QRS_NEXT_CUT()
PTP {E1 29336.909,E2 29336.909}
PTP {X 0,Y 607.909,A -85,B 0,C 180,E1 29336.909,E2 29336.909,E3 0,E4 0,E5 0,E6 0}
QRS_SPEED_INIT()
LIN {X 0,Y 607.909,Z 550,A -85,B 0,C 180,E1 29336.909,E2 29336.909,E3 0,E4 0,E5 0,E6 0} C_VEL
LIN {X 0,Y 607.909,Z 56.154,A -85,B 0,C 180,E1 29336.909,E2 29336.909} C_VEL
LIN {X 0,Y 607.909,Z 48.076,A -85,B 0,C 180,E1 29336.909,E2 29336.909} C_VEL
LIN {X 0,Y 607.891,Z 46.076,A -85,B 0,C 180,E1 29336.721,E2 29336.721} C_VEL
LIN {X 0,Y 607.912,Z 46.07,A -85,B 0,C 180,E1 29333.578,E2 29333.578} C_VEL
LIN {X 0,Y 607.871,Z 46.073,A -85,B 0,C 180,E1 29330.437,E2 29330.437} C_VEL
LIN {X 0,Y 607.918,Z 46.076,A -85,B 0,C 180,E1 29327.268,E2 29327.268} C_VEL
LIN {X 0,Y 607.88,Z 46.071,A -85,B 0,C 180,E1 29324.154,E2 29324.154} C_VEL
LIN {X 0,Y 607.875,Z 46.075,A -85,B 0,C 180,E1 29320.893,E2 29320.893} C_VEL
LIN {X 0,Y 607.917,Z 46.071,A -85,B 0,C 180,E1 29317.772,E2 29317.772} C_VEL
LIN {X 0,Y 607.864,Z 46.073,A -85,B 0,C 180,E1 29314.68,E2 29314.68} C_VEL
LIN {X 0,Y 607.915,Z 46.077,A -85,B 0,C 180,E1 29311.619,E2 29311.619} C_VEL
LIN {X 0,Y 607.867,Z 46.073,A -85,B 0,C 180,E1 29308.572,E2 29308.572} C_VEL
LIN {X 0,Y 607.874,Z 46.076,A -85,B 0,C 180,E1 29305.311,E2 29305.311} C_VEL
LIN {X 0,Y 607.9,Z 46.072,A -85,B 0,C 180,E1 29302.276,E2 29302.276} C_VEL
LIN {X 0,Y 607.858,Z 46.075,A -85,B 0,C 180,E1 29299.167,E2 29299.167} C_VEL
LIN {X 0,Y 607.917,Z 46.075,A -85,B 0,C 180,E1 29296.046,E2 29296.046} C_VEL
LIN {X 0,Y 607.854,Z 46.074,A -85,B 0,C 180,E1 29293.048,E2 29293.048} C_VEL
LIN {X 0,Y 607.895,Z 46.077,A -85,B 0,C 180,E1 29289.9,E2 29289.9} C_VEL
LIN {X 0,Y 607.862,Z 46.075,A -85,B 0,C 180,E1 29286.896,E2 29286.896} C_VEL
LIN {X 0,Y 607.859,Z 46.077,A -85,B 0,C 180,E1 29283.662,E2 29283.662} C_VEL
LIN {X 0,Y 607.917,Z 46.319,A -85,B 0,C 180,E1 29282.298,E2 29282.298} C_VEL
LIN {X 0,Y 607.876,Z 75.31,A -85,B 0,C 180,E1 29279.242,E2 29279.242} C_VEL
LIN {X 0,Y 607.896,Z 105.548,A -85,B 0,C 180,E1 29276.096,E2 29276.096} C_VEL
LIN {X 0,Y 607.888,Z 135.983,A -85,B 0,C 180,E1 29272.993,E2 29272.993} C_VEL
LIN {X 0,Y 607.857,Z 167.849,A -85,B 0,C 180,E1 29269.799,E2 29269.799} C_VEL
LIN {X 0,Y 607.909,Z 175.996,A -85,B 0,C 180,E1 29269.017,E2 29269.017} C_VEL
LIN {X 0,Y 607.889,Z 287.389,A -85,B 0,C 180,E1 29267.665,E2 29267.665} C_VEL
LIN {X 0,Y 607.914,Z 301.952,A -85,B 0,C 180,E1 29267.318,E2 29267.318} C_VEL
LIN {X 0,Y 607.92,Z 316.749,A -85,B 0,C 180,E1 29266.772,E2 29266.772} C_VEL
LIN {X 0,Y 607.887,Z 330.107,A -85,B 0,C 180,E1 29266.089,E2 29266.089} C_VEL
LIN {X 0,Y 607.919,Z 342.573,A -85,B 0,C 180,E1 29265.256,E2 29265.256} C_VEL
LIN {X 0,Y 607.918,Z 354.434,A -85,B 0,C 180,E1 29264.233,E2 29264.233} C_VEL
LIN {X 0,Y 607.918,Z 364.498,A -85,B 0,C 180,E1 29263.118,E2 29263.118} C_VEL
LIN {X 0,Y 607.918,Z 372.672,A -85,B 0,C 180,E1 29261.959,E2 29261.959} C_VEL
LIN {X 0,Y 607.916,Z 379.43,A -85,B 0,C 180,E1 29260.71,E2 29260.71} C_VEL
LIN {X 0,Y 607.917,Z 384.633,A -85,B 0,C 180,E1 29259.37,E2 29259.37} C_VEL
LIN {X 0,Y 607.917,Z 388.043,A -85,B 0,C 180,E1 29258.036,E2 29258.036} C_VEL
LIN {X 0,Y 607.916,Z 389.855,A -85,B 0,C 180,E1 29256.516,E2 29256.516} C_VEL
LIN {X 0,Y 607.916,Z 389.644,A -85,B 0,C 180,E1 29255.095,E2 29255.095} C_VEL
LIN {X 0,Y 607.917,Z 387.832,A -85,B 0,C 180,E1 29253.771,E2 29253.771} C_VEL
LIN {X 0,Y 607.915,Z 384.046,A -85,B 0,C 180,E1 29252.356,E2 29252.356} C_VEL
LIN {X 0,Y 607.916,Z 378.633,A -85,B 0,C 180,E1 29251.036,E2 29251.036} C_VEL
LIN {X 0,Y 607.918,Z 371.814,A -85,B 0,C 180,E1 29249.811,E2 29249.811} C_VEL
LIN {X 0,Y 607.917,Z 362.817,A -85,B 0,C 180,E1 29248.586,E2 29248.586} C_VEL
LIN {X 0,Y 607.919,Z 352.577,A -85,B 0,C 180,E1 29247.501,E2 29247.501} C_VEL
LIN {X 0,Y 607.916,Z 341.267,A -85,B 0,C 180,E1 29246.558,E2 29246.558} C_VEL
LIN {X 0,Y 607.886,Z 328.997,A -85,B 0,C 180,E1 29245.755,E2 29245.755} C_VEL
LIN {X 0,Y 607.919,Z 315.694,A -85,B 0,C 180,E1 29245.093,E2 29245.093} C_VEL
LIN {X 0,Y 607.871,Z 301.315,A -85,B 0,C 180,E1 29244.572,E2 29244.572} C_VEL
LIN {X 0,Y 607.846,Z 285.893,A -85,B 0,C 180,E1 29244.217,E2 29244.217} C_VEL
LIN {X 0,Y 607.887,Z 172.229,A -85,B 0,C 180,E1 29242.842,E2 29242.842} C_VEL
LIN {X 0,Y 607.851,Z 122.898,A -85,B 0,C 180,E1 29239.91,E2 29239.91} C_VEL
LIN {X 0,Y 607.917,Z 72.713,A -85,B 0,C 180,E1 29236.881,E2 29236.881} C_VEL
LIN {X 0,Y 607.911,Z 46.445,A -85,B 0,C 180,E1 29235.248,E2 29235.248} C_VEL
LIN {X 0,Y 607.873,Z 46.078,A -85,B 0,C 180,E1 29234.741,E2 29234.741} C_VEL
LIN {X 0,Y 607.903,Z 46.075,A -85,B 0,C 180,E1 29231.69,E2 29231.69} C_VEL
LIN {X 0,Y 607.917,Z 46.394,A -85,B 0,C 180,E1 29230.67,E2 29230.67} C_VEL
LIN {X 0,Y 607.919,Z 77.534,A -85,B 0,C 180,E1 29228.736,E2 29228.736} C_VEL
LIN {X 0,Y 607.908,Z 131.003,A -85,B 0,C 180,E1 29225.513,E2 29225.513} C_VEL
LIN {X 0,Y 607.913,Z 172.508,A -85,B 0,C 180,E1 29223.057,E2 29223.057} C_VEL
LIN {X 0,Y 607.898,Z 286.479,A -85,B 0,C 180,E1 29221.681,E2 29221.681} C_VEL
LIN {X 0,Y 607.915,Z 301.764,A -85,B 0,C 180,E1 29221.324,E2 29221.324} C_VEL
LIN {X 0,Y 607.919,Z 315.969,A -85,B 0,C 180,E1 29220.805,E2 29220.805} C_VEL
LIN {X 0,Y 607.892,Z 328.884,A -85,B 0,C 180,E1 29220.162,E2 29220.162} C_VEL
LIN {X 0,Y 607.92,Z 342.165,A -85,B 0,C 180,E1 29219.287,E2 29219.287} C_VEL
LIN {X 0,Y 607.918,Z 353.72,A -85,B 0,C 180,E1 29218.301,E2 29218.301} C_VEL
LIN {X 0,Y 607.918,Z 363.5,A -85,B 0,C 180,E1 29217.24,E2 29217.24} C_VEL
LIN {X 0,Y 607.918,Z 371.729,A -85,B 0,C 180,E1 29216.112,E2 29216.112} C_VEL
LIN {X 0,Y 607.918,Z 378.852,A -85,B 0,C 180,E1 29214.829,E2 29214.829} C_VEL
LIN {X 0,Y 607.918,Z 384.09,A -85,B 0,C 180,E1 29213.541,E2 29213.541} C_VEL
LIN {X 0,Y 607.917,Z 387.837,A -85,B 0,C 180,E1 29212.137,E2 29212.137} C_VEL
LIN {X 0,Y 607.919,Z 389.717,A -85,B 0,C 180,E1 29210.712,E2 29210.712} C_VEL
LIN {X 0,Y 607.916,Z 389.794,A -85,B 0,C 180,E1 29209.308,E2 29209.308} C_VEL
LIN {X 0,Y 607.915,Z 388.001,A -85,B 0,C 180,E1 29207.852,E2 29207.852} C_VEL
LIN {X 0,Y 607.915,Z 384.307,A -85,B 0,C 180,E1 29206.438,E2 29206.438} C_VEL
LIN {X 0,Y 607.918,Z 379.055,A -85,B 0,C 180,E1 29205.123,E2 29205.123} C_VEL
LIN {X 0,Y 607.917,Z 371.895,A -85,B 0,C 180,E1 29203.823,E2 29203.823} C_VEL
LIN {X 0,Y 607.918,Z 362.918,A -85,B 0,C 180,E1 29202.598,E2 29202.598} C_VEL
LIN {X 0,Y 607.918,Z 352.733,A -85,B 0,C 180,E1 29201.516,E2 29201.516} C_VEL
LIN {X 0,Y 607.92,Z 341.77,A -85,B 0,C 180,E1 29200.594,E2 29200.594} C_VEL
LIN {X 0,Y 607.916,Z 328.454,A -85,B 0,C 180,E1 29199.724,E2 29199.724} C_VEL
LIN {X 0,Y 607.919,Z 314.572,A -85,B 0,C 180,E1 29199.045,E2 29199.045} C_VEL
LIN {X 0,Y 607.914,Z 300.906,A -85,B 0,C 180,E1 29198.562,E2 29198.562} C_VEL
LIN {X 0,Y 607.908,Z 285.815,A -85,B 0,C 180,E1 29198.217,E2 29198.217} C_VEL
LIN {X 0,Y 607.916,Z 175.701,A -85,B 0,C 180,E1 29196.879,E2 29196.879} C_VEL
LIN {X 0,Y 607.918,Z 143.97,A -85,B 0,C 180,E1 29193.723,E2 29193.723} C_VEL
LIN {X 0,Y 607.892,Z 112.689,A -85,B 0,C 180,E1 29190.547,E2 29190.547} C_VEL
LIN {X 0,Y 607.897,Z 82.49,A -85,B 0,C 180,E1 29187.422,E2 29187.422} C_VEL
LIN {X 0,Y 607.918,Z 53.339,A -85,B 0,C 180,E1 29184.332,E2 29184.332} C_VEL
LIN {X 0,Y 607.901,Z 46.197,A -85,B 0,C 180,E1 29183.507,E2 29183.507} C_VEL
LIN {X 0,Y 607.882,Z 46.072,A -85,B 0,C 180,E1 29180.509,E2 29180.509} C_VEL
LIN {X 0,Y 607.872,Z 46.075,A -85,B 0,C 180,E1 29177.321,E2 29177.321} C_VEL
LIN {X 0,Y 607.918,Z 46.072,A -85,B 0,C 180,E1 29174.186,E2 29174.186} C_VEL
LIN {X 0,Y 607.861,Z 46.074,A -85,B 0,C 180,E1 29171.096,E2 29171.096} C_VEL
LIN {X 0,Y 607.908,Z 46.077,A -85,B 0,C 180,E1 29167.942,E2 29167.942} C_VEL
LIN {X 0,Y 607.867,Z 46.074,A -85,B 0,C 180,E1 29164.907,E2 29164.907} C_VEL
LIN {X 0,Y 607.862,Z 46.076,A -85,B 0,C 180,E1 29161.603,E2 29161.603} C_VEL
LIN {X 0,Y 607.906,Z 46.073,A -85,B 0,C 180,E1 29158.586,E2 29158.586} C_VEL
LIN {X 0,Y 607.852,Z 46.075,A -85,B 0,C 180,E1 29155.472,E2 29155.472} C_VEL
LIN {X 0,Y 607.919,Z 46.077,A -85,B 0,C 180,E1 29152.439,E2 29152.439} C_VEL
LIN {X 0,Y 607.852,Z 46.075,A -85,B 0,C 180,E1 29149.384,E2 29149.384} C_VEL
LIN {X 0,Y 607.876,Z 46.077,A -85,B 0,C 180,E1 29146.202,E2 29146.202} C_VEL
LIN {X 0,Y 607.861,Z 46.075,A -85,B 0,C 180,E1 29143.271,E2 29143.271} C_VEL
LIN {X 0,Y 607.854,Z 46.076,A -85,B 0,C 180,E1 29140.093,E2 29140.093} C_VEL
LIN {X 0,Y 607.88,Z 46.075,A -85,B 0,C 180,E1 29137.159,E2 29137.159} C_VEL
LIN {X 0,Y 607.843,Z 46.077,A -85,B 0,C 180,E1 29134.052,E2 29134.052} C_VEL
LIN {X 0,Y 607.904,Z 46.076,A -85,B 0,C 180,E1 29131.046,E2 29131.046} C_VEL
LIN {X 0,Y 607.837,Z 46.077,A -85,B 0,C 180,E1 29128.017,E2 29128.017} C_VEL
LIN {X 0,Y 607.908,Z 46.077,A -85,B 0,C 180,E1 29124.969,E2 29124.969} C_VEL
LIN {X 0,Y 607.834,Z 46.077,A -85,B 0,C 180,E1 29121.993,E2 29121.993} C_VEL
LIN {X 0,Y 607.871,Z 46.078,A -85,B 0,C 180,E1 29118.857,E2 29118.857} C_VEL
LIN {X 0,Y 607.836,Z 46.077,A -85,B 0,C 180,E1 29116.039,E2 29116.039} C_VEL
LIN {X 0,Y 607.868,Z 46.077,A -85,B 0,C 180,E1 29112.92,E2 29112.92} C_VEL
LIN {X 0,Y 607.842,Z 46.077,A -85,B 0,C 180,E1 29110.103,E2 29110.103} C_VEL
LIN {X 0,Y 607.858,Z 46.076,A -85,B 0,C 180,E1 29106.898,E2 29106.898} C_VEL
LIN {X 0,Y 607.86,Z 46.077,A -85,B 0,C 180,E1 29104.002,E2 29104.002} C_VEL
LIN {X 0,Y 607.849,Z 46.079,A -85,B 0,C 180,E1 29100.835,E2 29100.835} C_VEL
LIN {X 0,Y 607.894,Z 46.318,A -85,B 0,C 180,E1 29099.784,E2 29099.784} C_VEL
LIN {X 0,Y 607.919,Z 52.934,A -85,B 0,C 180,E1 29099.292,E2 29099.292} C_VEL
LIN {X 0,Y 607.902,Z 98.568,A -85,B 0,C 180,E1 29096.208,E2 29096.208} C_VEL
LIN {X 0,Y 607.909,Z 145.038,A -85,B 0,C 180,E1 29093.148,E2 29093.148} C_VEL
LIN {X 0,Y 607.901,Z 157.996,A -85,B 0,C 180,E1 29092.33,E2 29092.33} C_VEL
LIN {X 0,Y 607.917,Z 367.301,A -85,B 0,C 180,E1 29089.705,E2 29089.705} C_VEL
LIN {X 0,Y 607.914,Z 385.58,A -85,B 0,C 180,E1 29089.305,E2 29089.305} C_VEL
LIN {X 0,Y 607.912,Z 404.399,A -85,B 0,C 180,E1 29088.707,E2 29088.707} C_VEL
LIN {X 0,Y 607.915,Z 422.05,A -85,B 0,C 180,E1 29087.963,E2 29087.963} C_VEL
LIN {X 0,Y 607.919,Z 438.783,A -85,B 0,C 180,E1 29087.073,E2 29087.073} C_VEL
LIN {X 0,Y 607.916,Z 454.637,A -85,B 0,C 180,E1 29086.041,E2 29086.041} C_VEL
LIN {X 0,Y 607.917,Z 469.558,A -85,B 0,C 180,E1 29084.868,E2 29084.868} C_VEL
LIN {X 0,Y 607.918,Z 483.217,A -85,B 0,C 180,E1 29083.583,E2 29083.583} C_VEL
LIN {X 0,Y 607.916,Z 495.903,A -85,B 0,C 180,E1 29082.154,E2 29082.154} C_VEL
LIN {X 0,Y 607.912,Z 507.221,A -85,B 0,C 180,E1 29080.616,E2 29080.616} C_VEL
LIN {X 0,Y 607.918,Z 516.986,A -85,B 0,C 180,E1 29078.99,E2 29078.99} C_VEL
LIN {X 0,Y 607.91,Z 524.861,A -85,B 0,C 180,E1 29077.35,E2 29077.35} C_VEL
LIN {X 0,Y 607.907,Z 531.106,A -85,B 0,C 180,E1 29075.664,E2 29075.664} C_VEL
LIN {X 0,Y 607.916,Z 535.871,A -85,B 0,C 180,E1 29073.867,E2 29073.867} C_VEL
LIN {X 0,Y 607.914,Z 538.786,A -85,B 0,C 180,E1 29072.074,E2 29072.074} C_VEL
LIN {X 0,Y 607.907,Z 539.939,A -85,B 0,C 180,E1 29070.283,E2 29070.283} C_VEL
LIN {X 0,Y 607.916,Z 539.348,A -85,B 0,C 180,E1 29068.493,E2 29068.493} C_VEL
LIN {X 0,Y 607.908,Z 537.006,A -85,B 0,C 180,E1 29066.701,E2 29066.701} C_VEL
LIN {X 0,Y 607.916,Z 533.098,A -85,B 0,C 180,E1 29065,E2 29065} C_VEL
LIN {X 0,Y 607.91,Z 527.47,A -85,B 0,C 180,E1 29063.295,E2 29063.295} C_VEL
LIN {X 0,Y 607.915,Z 520.426,A -85,B 0,C 180,E1 29061.679,E2 29061.679} C_VEL
LIN {X 0,Y 607.912,Z 511.514,A -85,B 0,C 180,E1 29060.056,E2 29060.056} C_VEL
LIN {X 0,Y 607.919,Z 501.151,A -85,B 0,C 180,E1 29058.522,E2 29058.522} C_VEL
LIN {X 0,Y 607.917,Z 489.353,A -85,B 0,C 180,E1 29057.076,E2 29057.076} C_VEL
LIN {X 0,Y 607.915,Z 476.098,A -85,B 0,C 180,E1 29055.718,E2 29055.718} C_VEL
LIN {X 0,Y 607.917,Z 461.246,A -85,B 0,C 180,E1 29054.45,E2 29054.45} C_VEL
LIN {X 0,Y 607.918,Z 445.235,A -85,B 0,C 180,E1 29053.322,E2 29053.322} C_VEL
LIN {X 0,Y 607.913,Z 429.047,A -85,B 0,C 180,E1 29052.385,E2 29052.385} C_VEL
LIN {X 0,Y 607.914,Z 412.089,A -85,B 0,C 180,E1 29051.593,E2 29051.593} C_VEL
LIN {X 0,Y 607.914,Z 394.258,A -85,B 0,C 180,E1 29050.946,E2 29050.946} C_VEL
LIN {X 0,Y 607.916,Z 375.204,A -85,B 0,C 180,E1 29050.447,E2 29050.447} C_VEL
LIN {X 0,Y 607.916,Z 355.852,A -85,B 0,C 180,E1 29050.129,E2 29050.129} C_VEL
LIN {X 0,Y 607.897,Z 154.774,A -85,B 0,C 180,E1 29047.622,E2 29047.622} C_VEL
LIN {X 0,Y 607.918,Z 76.627,A -85,B 0,C 180,E1 29044.58,E2 29044.58} C_VEL
LIN {X 0,Y 607.913,Z 46.741,A -85,B 0,C 180,E1 29043.374,E2 29043.374} C_VEL
LIN {X 0,Y 607.903,Z 46.125,A -85,B 0,C 180,E1 29043.215,E2 29043.215} C_VEL
LIN {X 0,Y 607.899,Z 46.073,A -85,B 0,C 180,E1 29040.001,E2 29040.001} C_VEL
LIN {X 0,Y 607.9,Z 46.069,A -85,B 0,C 180,E1 29036.845,E2 29036.845} C_VEL
LIN {X 0,Y 607.911,Z 46.076,A -85,B 0,C 180,E1 29033.578,E2 29033.578} C_VEL
LIN {X 0,Y 607.903,Z 46.071,A -85,B 0,C 180,E1 29030.331,E2 29030.331} C_VEL
LIN {X 0,Y 607.893,Z 46.071,A -85,B 0,C 180,E1 29027.187,E2 29027.187} C_VEL
LIN {X 0,Y 607.916,Z 46.077,A -85,B 0,C 180,E1 29023.954,E2 29023.954} C_VEL
LIN {X 0,Y 607.912,Z 46.068,A -85,B 0,C 180,E1 29020.694,E2 29020.694} C_VEL
LIN {X 0,Y 607.889,Z 46.072,A -85,B 0,C 180,E1 29017.487,E2 29017.487} C_VEL
LIN {X 0,Y 607.908,Z 46.074,A -85,B 0,C 180,E1 29014.343,E2 29014.343} C_VEL
LIN {X 0,Y 607.898,Z 46.069,A -85,B 0,C 180,E1 29011.205,E2 29011.205} C_VEL
LIN {X 0,Y 607.894,Z 46.075,A -85,B 0,C 180,E1 29007.954,E2 29007.954} C_VEL
LIN {X 0,Y 607.908,Z 46.071,A -85,B 0,C 180,E1 29004.787,E2 29004.787} C_VEL
LIN {X 0,Y 607.884,Z 46.072,A -85,B 0,C 180,E1 29001.675,E2 29001.675} C_VEL
LIN {X 0,Y 607.919,Z 46.077,A -85,B 0,C 180,E1 28998.508,E2 28998.508} C_VEL
LIN {X 0,Y 607.916,Z 46.068,A -85,B 0,C 180,E1 28995.257,E2 28995.257} C_VEL
LIN {X 0,Y 607.88,Z 46.073,A -85,B 0,C 180,E1 28992.057,E2 28992.057} C_VEL
LIN {X 0,Y 607.913,Z 46.074,A -85,B 0,C 180,E1 28988.894,E2 28988.894} C_VEL
LIN {X 0,Y 607.887,Z 46.07,A -85,B 0,C 180,E1 28985.758,E2 28985.758} C_VEL
LIN {X 0,Y 607.883,Z 46.075,A -85,B 0,C 180,E1 28982.451,E2 28982.451} C_VEL
LIN {X 0,Y 607.914,Z 46.071,A -85,B 0,C 180,E1 28979.34,E2 28979.34} C_VEL
LIN {X 0,Y 607.891,Z 46.076,A -85,B 0,C 180,E1 28976.721,E2 28976.721} C_VEL
LIN {X 0,Y 606.874,Z 46.2,A -85,B 0,C 180,E1 28975.995,E2 28975.995} C_VEL
LIN {X 0,Y 600.5,Z 46.993,A -85,B 0,C 180,E1 28973.958,E2 28973.958} C_VEL
LIN {X 0,Y 599.976,Z 47.06,A -85,B 0,C 180,E1 28973.428,E2 28973.428} C_VEL
LIN {X 0,Y 599.933,Z 47.061,A -85,B 0,C 180,E1 28970.309,E2 28970.309} C_VEL
LIN {X 0,Y 599.964,Z 47.065,A -85,B 0,C 180,E1 28967.096,E2 28967.096} C_VEL
LIN {X 0,Y 599.96,Z 47.059,A -85,B 0,C 180,E1 28963.94,E2 28963.94} C_VEL
LIN {X 0,Y 599.93,Z 47.063,A -85,B 0,C 180,E1 28960.731,E2 28960.731} C_VEL
LIN {X 0,Y 599.978,Z 47.064,A -85,B 0,C 180,E1 28957.565,E2 28957.565} C_VEL
LIN {X 0,Y 599.933,Z 47.061,A -85,B 0,C 180,E1 28954.427,E2 28954.427} C_VEL
LIN {X 0,Y 599.932,Z 47.063,A -85,B 0,C 180,E1 28951.097,E2 28951.097} C_VEL
LIN {X 0,Y 599.977,Z 47.06,A -85,B 0,C 180,E1 28947.998,E2 28947.998} C_VEL
LIN {X 0,Y 599.921,Z 47.062,A -85,B 0,C 180,E1 28944.9,E2 28944.9} C_VEL
LIN {X 0,Y 599.964,Z 47.066,A -85,B 0,C 180,E1 28941.687,E2 28941.687} C_VEL
LIN {X 0,Y 599.936,Z 47.062,A -85,B 0,C 180,E1 28938.574,E2 28938.574} C_VEL
LIN {X 0,Y 599.922,Z 47.065,A -85,B 0,C 180,E1 28935.368,E2 28935.368} C_VEL
LIN {X 0,Y 599.976,Z 47.062,A -85,B 0,C 180,E1 28932.274,E2 28932.274} C_VEL
LIN {X 0,Y 599.913,Z 47.064,A -85,B 0,C 180,E1 28929.172,E2 28929.172} C_VEL
LIN {X 0,Y 599.961,Z 47.067,A -85,B 0,C 180,E1 28926.034,E2 28926.034} C_VEL
LIN {X 0,Y 599.919,Z 47.067,A -85,B 0,C 180,E1 28923.023,E2 28923.023} C_VEL
LIN {X 0,Y 600.016,Z 47.343,A -85,B 0,C 180,E1 28922.435,E2 28922.435} C_VEL
LIN {X 0,Y 600.181,Z 73.388,A -85,B 0,C 180,E1 28919.764,E2 28919.764} C_VEL
LIN {X 0,Y 600.158,Z 103.091,A -85,B 0,C 180,E1 28916.624,E2 28916.624} C_VEL
LIN {X 0,Y 600.06,Z 133.601,A -85,B 0,C 180,E1 28913.467,E2 28913.467} C_VEL
LIN {X 0,Y 599.995,Z 164.422,A -85,B 0,C 180,E1 28910.331,E2 28910.331} C_VEL
LIN {X 0,Y 600.046,Z 176.097,A -85,B 0,C 180,E1 28909.187,E2 28909.187} C_VEL
LIN {X 0,Y 600.052,Z 287.645,A -85,B 0,C 180,E1 28907.816,E2 28907.816} C_VEL
LIN {X 0,Y 600.057,Z 302.488,A -85,B 0,C 180,E1 28907.452,E2 28907.452} C_VEL
LIN {X 0,Y 600.04,Z 317.043,A -85,B 0,C 180,E1 28906.903,E2 28906.903} C_VEL
LIN {X 0,Y 599.98,Z 330.388,A -85,B 0,C 180,E1 28906.208,E2 28906.208} C_VEL
LIN {X 0,Y 599.984,Z 342.784,A -85,B 0,C 180,E1 28905.364,E2 28905.364} C_VEL
LIN {X 0,Y 599.96,Z 354.596,A -85,B 0,C 180,E1 28904.328,E2 28904.328} C_VEL
LIN {X 0,Y 599.943,Z 364.632,A -85,B 0,C 180,E1 28903.197,E2 28903.197} C_VEL
LIN {X 0,Y 599.929,Z 372.773,A -85,B 0,C 180,E1 28902.023,E2 28902.023} C_VEL
LIN {X 0,Y 599.922,Z 379.505,A -85,B 0,C 180,E1 28900.757,E2 28900.757} C_VEL
LIN {X 0,Y 599.918,Z 384.791,A -85,B 0,C 180,E1 28899.366,E2 28899.366} C_VEL
LIN {X 0,Y 599.917,Z 388.072,A -85,B 0,C 180,E1 28898.047,E2 28898.047} C_VEL
LIN {X 0,Y 599.916,Z 389.865,A -85,B 0,C 180,E1 28896.507,E2 28896.507} C_VEL
LIN {X 0,Y 599.916,Z 389.633,A -85,B 0,C 180,E1 28895.067,E2 28895.067} C_VEL
LIN {X 0,Y 599.916,Z 387.798,A -85,B 0,C 180,E1 28893.726,E2 28893.726} C_VEL
LIN {X 0,Y 599.917,Z 383.997,A -85,B 0,C 180,E1 28892.292,E2 28892.292} C_VEL
LIN {X 0,Y 599.922,Z 378.559,A -85,B 0,C 180,E1 28890.954,E2 28890.954} C_VEL
LIN {X 0,Y 599.932,Z 371.709,A -85,B 0,C 180,E1 28889.713,E2 28889.713} C_VEL
LIN {X 0,Y 599.944,Z 362.694,A -85,B 0,C 180,E1 28888.471,E2 28888.471} C_VEL
LIN {X 0,Y 599.964,Z 352.416,A -85,B 0,C 180,E1 28887.373,E2 28887.373} C_VEL
LIN {X 0,Y 599.981,Z 341.056,A -85,B 0,C 180,E1 28886.416,E2 28886.416} C_VEL
LIN {X 0,Y 599.983,Z 328.728,A -85,B 0,C 180,E1 28885.603,E2 28885.603} C_VEL
LIN {X 0,Y 600.041,Z 315.333,A -85,B 0,C 180,E1 28884.933,E2 28884.933} C_VEL
LIN {X 0,Y 600.017,Z 301.58,A -85,B 0,C 180,E1 28884.429,E2 28884.429} C_VEL
LIN {X 0,Y 600.01,Z 285.975,A -85,B 0,C 180,E1 28884.063,E2 28884.063} C_VEL
LIN {X 0,Y 600.047,Z 172.413,A -85,B 0,C 180,E1 28882.676,E2 28882.676} C_VEL
LIN {X 0,Y 600.081,Z 123.44,A -85,B 0,C 180,E1 28879.73,E2 28879.73} C_VEL
LIN {X 0,Y 600.237,Z 74.053,A -85,B 0,C 180,E1 28876.71,E2 28876.71} C_VEL
LIN {X 0,Y 600.139,Z 48.039,A -85,B 0,C 180,E1 28875.086,E2 28875.086} C_VEL
LIN {X 0,Y 599.953,Z 47.121,A -85,B 0,C 180,E1 28874.93,E2 28874.93} C_VEL
LIN {X 0,Y 599.964,Z 47.065,A -85,B 0,C 180,E1 28871.792,E2 28871.792} C_VEL
LIN {X 0,Y 599.99,Z 47.204,A -85,B 0,C 180,E1 28870.935,E2 28870.935} C_VEL
LIN {X 0,Y 600.288,Z 49.166,A -85,B 0,C 180,E1 28870.743,E2 28870.743} C_VEL
LIN {X 0,Y 600.187,Z 101.17,A -85,B 0,C 180,E1 28867.535,E2 28867.535} C_VEL
LIN {X 0,Y 600.062,Z 154.089,A -85,B 0,C 180,E1 28864.327,E2 28864.327} C_VEL
LIN {X 0,Y 600.108,Z 172.928,A -85,B 0,C 180,E1 28863.222,E2 28863.222} C_VEL
LIN {X 0,Y 600.062,Z 287.429,A -85,B 0,C 180,E1 28861.819,E2 28861.819} C_VEL
LIN {X 0,Y 600.061,Z 301.945,A -85,B 0,C 180,E1 28861.47,E2 28861.47} C_VEL
LIN {X 0,Y 600.039,Z 316.2,A -85,B 0,C 180,E1 28860.939,E2 28860.939} C_VEL
LIN {X 0,Y 599.984,Z 329.601,A -85,B 0,C 180,E1 28860.255,E2 28860.255} C_VEL
LIN {X 0,Y 599.985,Z 342.64,A -85,B 0,C 180,E1 28859.375,E2 28859.375} C_VEL
LIN {X 0,Y 599.96,Z 354.535,A -85,B 0,C 180,E1 28858.334,E2 28858.334} C_VEL
LIN {X 0,Y 599.942,Z 365.113,A -85,B 0,C 180,E1 28857.137,E2 28857.137} C_VEL
LIN {X 0,Y 599.93,Z 373.349,A -85,B 0,C 180,E1 28855.927,E2 28855.927} C_VEL
LIN {X 0,Y 599.923,Z 379.915,A -85,B 0,C 180,E1 28854.667,E2 28854.667} C_VEL
LIN {X 0,Y 599.919,Z 385.157,A -85,B 0,C 180,E1 28853.249,E2 28853.249} C_VEL
LIN {X 0,Y 599.916,Z 388.356,A -85,B 0,C 180,E1 28851.876,E2 28851.876} C_VEL
LIN {X 0,Y 599.916,Z 389.888,A -85,B 0,C 180,E1 28850.456,E2 28850.456} C_VEL
LIN {X 0,Y 599.914,Z 389.554,A -85,B 0,C 180,E1 28848.954,E2 28848.954} C_VEL
LIN {X 0,Y 599.917,Z 387.415,A -85,B 0,C 180,E1 28847.546,E2 28847.546} C_VEL
LIN {X 0,Y 599.919,Z 383.661,A -85,B 0,C 180,E1 28846.192,E2 28846.192} C_VEL
LIN {X 0,Y 599.924,Z 377.654,A -85,B 0,C 180,E1 28844.766,E2 28844.766} C_VEL
LIN {X 0,Y 599.932,Z 370.287,A -85,B 0,C 180,E1 28843.497,E2 28843.497} C_VEL
LIN {X 0,Y 599.947,Z 361.441,A -85,B 0,C 180,E1 28842.323,E2 28842.323} C_VEL
LIN {X 0,Y 599.969,Z 350.727,A -85,B 0,C 180,E1 28841.213,E2 28841.213} C_VEL
LIN {X 0,Y 599.981,Z 338.758,A -85,B 0,C 180,E1 28840.249,E2 28840.249} C_VEL
LIN {X 0,Y 600.014,Z 326.653,A -85,B 0,C 180,E1 28839.488,E2 28839.488} C_VEL
LIN {X 0,Y 600.045,Z 313.017,A -85,B 0,C 180,E1 28838.834,E2 28838.834} C_VEL
LIN {X 0,Y 600.064,Z 297.902,A -85,B 0,C 180,E1 28838.326,E2 28838.326} C_VEL
LIN {X 0,Y 600.076,Z 283.303,A -85,B 0,C 180,E1 28838.024,E2 28838.024} C_VEL
LIN {X 0,Y 600.03,Z 175.769,A -85,B 0,C 180,E1 28836.708,E2 28836.708} C_VEL
LIN {X 0,Y 600.074,Z 144.357,A -85,B 0,C 180,E1 28833.544,E2 28833.544} C_VEL
LIN {X 0,Y 600.127,Z 113.017,A -85,B 0,C 180,E1 28830.32,E2 28830.32} C_VEL
LIN {X 0,Y 600.201,Z 82.376,A -85,B 0,C 180,E1 28827.105,E2 28827.105} C_VEL
LIN {X 0,Y 600.381,Z 53.646,A -85,B 0,C 180,E1 28823.976,E2 28823.976} C_VEL
LIN {X 0,Y 600.154,Z 48.131,A -85,B 0,C 180,E1 28823.36,E2 28823.36} C_VEL
LIN {X 0,Y 599.942,Z 47.125,A -85,B 0,C 180,E1 28823.161,E2 28823.161} C_VEL
LIN {X 0,Y 599.978,Z 47.064,A -85,B 0,C 180,E1 28819.977,E2 28819.977} C_VEL
LIN {X 0,Y 599.927,Z 47.063,A -85,B 0,C 180,E1 28816.858,E2 28816.858} C_VEL
LIN {X 0,Y 599.956,Z 47.066,A -85,B 0,C 180,E1 28813.689,E2 28813.689} C_VEL
LIN {X 0,Y 599.951,Z 47.061,A -85,B 0,C 180,E1 28810.564,E2 28810.564} C_VEL
LIN {X 0,Y 599.922,Z 47.064,A -85,B 0,C 180,E1 28807.373,E2 28807.373} C_VEL
LIN {X 0,Y 599.979,Z 47.063,A -85,B 0,C 180,E1 28804.301,E2 28804.301} C_VEL
LIN {X 0,Y 599.917,Z 47.063,A -85,B 0,C 180,E1 28801.242,E2 28801.242} C_VEL
LIN {X 0,Y 599.957,Z 47.066,A -85,B 0,C 180,E1 28798.09,E2 28798.09} C_VEL
LIN {X 0,Y 599.93,Z 47.063,A -85,B 0,C 180,E1 28795.028,E2 28795.028} C_VEL
LIN {X 0,Y 599.917,Z 47.065,A -85,B 0,C 180,E1 28791.759,E2 28791.759} C_VEL
LIN {X 0,Y 599.978,Z 47.063,A -85,B 0,C 180,E1 28788.659,E2 28788.659} C_VEL
LIN {X 0,Y 599.908,Z 47.064,A -85,B 0,C 180,E1 28785.621,E2 28785.621} C_VEL
LIN {X 0,Y 599.969,Z 47.066,A -85,B 0,C 180,E1 28782.544,E2 28782.544} C_VEL
LIN {X 0,Y 599.911,Z 47.064,A -85,B 0,C 180,E1 28779.5,E2 28779.5} C_VEL
LIN {X 0,Y 599.915,Z 47.066,A -85,B 0,C 180,E1 28776.205,E2 28776.205} C_VEL
LIN {X 0,Y 599.937,Z 47.065,A -85,B 0,C 180,E1 28773.257,E2 28773.257} C_VEL
LIN {X 0,Y 599.901,Z 47.066,A -85,B 0,C 180,E1 28770.11,E2 28770.11} C_VEL
LIN {X 0,Y 599.968,Z 47.066,A -85,B 0,C 180,E1 28767.093,E2 28767.093} C_VEL
LIN {X 0,Y 599.896,Z 47.066,A -85,B 0,C 180,E1 28764.078,E2 28764.078} C_VEL
LIN {X 0,Y 599.963,Z 47.068,A -85,B 0,C 180,E1 28761.076,E2 28761.076} C_VEL
LIN {X 0,Y 599.893,Z 47.067,A -85,B 0,C 180,E1 28758.06,E2 28758.06} C_VEL
LIN {X 0,Y 599.937,Z 47.066,A -85,B 0,C 180,E1 28754.962,E2 28754.962} C_VEL
LIN {X 0,Y 599.902,Z 47.066,A -85,B 0,C 180,E1 28752.068,E2 28752.068} C_VEL
LIN {X 0,Y 599.913,Z 47.066,A -85,B 0,C 180,E1 28748.805,E2 28748.805} C_VEL
LIN {X 0,Y 599.926,Z 47.067,A -85,B 0,C 180,E1 28745.906,E2 28745.906} C_VEL
LIN {X 0,Y 599.909,Z 47.066,A -85,B 0,C 180,E1 28742.798,E2 28742.798} C_VEL
LIN {X 0,Y 599.945,Z 47.264,A -85,B 0,C 180,E1 28740.142,E2 28740.142} C_VEL
LIN {X 0,Y 600.606,Z 50.341,A -85,B 0,C 180,E1 28739.85,E2 28739.85} C_VEL
LIN {X 0,Y 600.513,Z 95.338,A -85,B 0,C 180,E1 28736.774,E2 28736.774} C_VEL
LIN {X 0,Y 600.378,Z 142.596,A -85,B 0,C 180,E1 28733.616,E2 28733.616} C_VEL
LIN {X 0,Y 600.408,Z 158.125,A -85,B 0,C 180,E1 28732.622,E2 28732.622} C_VEL
LIN {X 0,Y 600.377,Z 367.301,A -85,B 0,C 180,E1 28729.963,E2 28729.963} C_VEL
LIN {X 0,Y 600.334,Z 386.274,A -85,B 0,C 180,E1 28729.538,E2 28729.538} C_VEL
LIN {X 0,Y 600.284,Z 404.396,A -85,B 0,C 180,E1 28728.954,E2 28728.954} C_VEL
LIN {X 0,Y 600.23,Z 422.045,A -85,B 0,C 180,E1 28728.201,E2 28728.201} C_VEL
LIN {X 0,Y 600.179,Z 438.697,A -85,B 0,C 180,E1 28727.305,E2 28727.305} C_VEL
LIN {X 0,Y 600.121,Z 454.633,A -85,B 0,C 180,E1 28726.255,E2 28726.255} C_VEL
LIN {X 0,Y 600.069,Z 469.558,A -85,B 0,C 180,E1 28725.067,E2 28725.067} C_VEL
LIN {X 0,Y 600.022,Z 483.015,A -85,B 0,C 180,E1 28723.786,E2 28723.786} C_VEL
LIN {X 0,Y 599.982,Z 495.905,A -85,B 0,C 180,E1 28722.317,E2 28722.317} C_VEL
LIN {X 0,Y 599.954,Z 507.223,A -85,B 0,C 180,E1 28720.758,E2 28720.758} C_VEL
LIN {X 0,Y 599.935,Z 516.988,A -85,B 0,C 180,E1 28719.11,E2 28719.11} C_VEL
LIN {X 0,Y 599.921,Z 525.04,A -85,B 0,C 180,E1 28717.406,E2 28717.406} C_VEL
LIN {X 0,Y 599.911,Z 531.409,A -85,B 0,C 180,E1 28715.644,E2 28715.644} C_VEL
LIN {X 0,Y 599.915,Z 535.872,A -85,B 0,C 180,E1 28713.919,E2 28713.919} C_VEL
LIN {X 0,Y 599.914,Z 538.787,A -85,B 0,C 180,E1 28712.102,E2 28712.102} C_VEL
LIN {X 0,Y 599.907,Z 539.939,A -85,B 0,C 180,E1 28710.287,E2 28710.287} C_VEL
LIN {X 0,Y 599.915,Z 539.349,A -85,B 0,C 180,E1 28708.473,E2 28708.473} C_VEL
LIN {X 0,Y 599.907,Z 537.007,A -85,B 0,C 180,E1 28706.657,E2 28706.657} C_VEL
LIN {X 0,Y 599.917,Z 533.099,A -85,B 0,C 180,E1 28704.933,E2 28704.933} C_VEL
LIN {X 0,Y 599.919,Z 527.47,A -85,B 0,C 180,E1 28703.205,E2 28703.205} C_VEL
LIN {X 0,Y 599.929,Z 520.427,A -85,B 0,C 180,E1 28701.567,E2 28701.567} C_VEL
LIN {X 0,Y 599.942,Z 511.515,A -85,B 0,C 180,E1 28699.923,E2 28699.923} C_VEL
LIN {X 0,Y 599.969,Z 501.152,A -85,B 0,C 180,E1 28698.368,E2 28698.368} C_VEL
LIN {X 0,Y 600.002,Z 489.355,A -85,B 0,C 180,E1 28696.902,E2 28696.902} C_VEL
LIN {X 0,Y 600.046,Z 475.762,A -85,B 0,C 180,E1 28695.494,E2 28695.494} C_VEL
LIN {X 0,Y 600.103,Z 461.244,A -85,B 0,C 180,E1 28694.243,E2 28694.243} C_VEL
LIN {X 0,Y 600.165,Z 445.239,A -85,B 0,C 180,E1 28693.1,E2 28693.1} C_VEL
LIN {X 0,Y 600.219,Z 428.058,A -85,B 0,C 180,E1 28692.102,E2 28692.102} C_VEL
LIN {X 0,Y 600.278,Z 410.698,A -85,B 0,C 180,E1 28691.295,E2 28691.295} C_VEL
LIN {X 0,Y 600.329,Z 392.689,A -85,B 0,C 180,E1 28690.649,E2 28690.649} C_VEL
LIN {X 0,Y 600.368,Z 374.196,A -85,B 0,C 180,E1 28690.172,E2 28690.172} C_VEL
LIN {X 0,Y 600.391,Z 354.456,A -85,B 0,C 180,E1 28689.852,E2 28689.852} C_VEL
LIN {X 0,Y 600.442,Z 154.702,A -85,B 0,C 180,E1 28687.327,E2 28687.327} C_VEL
LIN {X 0,Y 600.604,Z 75.307,A -85,B 0,C 180,E1 28684.195,E2 28684.195} C_VEL
LIN {X 0,Y 600.647,Z 49.473,A -85,B 0,C 180,E1 28683.157,E2 28683.157} C_VEL
LIN {X 0,Y 600.013,Z 47.428,A -85,B 0,C 180,E1 28683,E2 28683} C_VEL
LIN {X 0,Y 599.973,Z 47.062,A -85,B 0,C 180,E1 28682.402,E2 28682.402} C_VEL
LIN {X 0,Y 599.958,Z 47.062,A -85,B 0,C 180,E1 28679.123,E2 28679.123} C_VEL
LIN {X 0,Y 599.964,Z 47.063,A -85,B 0,C 180,E1 28675.921,E2 28675.921} C_VEL
LIN {X 0,Y 599.973,Z 47.057,A -85,B 0,C 180,E1 28672.648,E2 28672.648} C_VEL
LIN {X 0,Y 599.959,Z 47.063,A -85,B 0,C 180,E1 28669.459,E2 28669.459} C_VEL
LIN {X 0,Y 599.965,Z 47.062,A -85,B 0,C 180,E1 28666.244,E2 28666.244} C_VEL
LIN {X 0,Y 599.958,Z 47.059,A -85,B 0,C 180,E1 28663.101,E2 28663.101} C_VEL
LIN {X 0,Y 599.963,Z 47.064,A -85,B 0,C 180,E1 28659.788,E2 28659.788} C_VEL
LIN {X 0,Y 599.966,Z 47.06,A -85,B 0,C 180,E1 28656.56,E2 28656.56} C_VEL
LIN {X 0,Y 599.951,Z 47.06,A -85,B 0,C 180,E1 28653.392,E2 28653.392} C_VEL
LIN {X 0,Y 599.97,Z 47.066,A -85,B 0,C 180,E1 28650.129,E2 28650.129} C_VEL
LIN {X 0,Y 599.971,Z 47.058,A -85,B 0,C 180,E1 28646.848,E2 28646.848} C_VEL
LIN {X 0,Y 599.945,Z 47.06,A -85,B 0,C 180,E1 28643.681,E2 28643.681} C_VEL
LIN {X 0,Y 599.978,Z 47.066,A -85,B 0,C 180,E1 28640.485,E2 28640.485} C_VEL
LIN {X 0,Y 599.978,Z 47.057,A -85,B 0,C 180,E1 28637.156,E2 28637.156} C_VEL
LIN {X 0,Y 599.942,Z 47.062,A -85,B 0,C 180,E1 28633.984,E2 28633.984} C_VEL
LIN {X 0,Y 599.975,Z 47.065,A -85,B 0,C 180,E1 28630.757,E2 28630.757} C_VEL
LIN {X 0,Y 599.968,Z 47.058,A -85,B 0,C 180,E1 28627.469,E2 28627.469} C_VEL
LIN {X 0,Y 599.941,Z 47.062,A -85,B 0,C 180,E1 28624.301,E2 28624.301} C_VEL
LIN {X 0,Y 599.974,Z 47.062,A -85,B 0,C 180,E1 28621.146,E2 28621.146} C_VEL
LIN {X 0,Y 599.941,Z 47.06,A -85,B 0,C 180,E1 28617.994,E2 28617.994} C_VEL
LIN {X 0,Y 599.95,Z 47.064,A -85,B 0,C 180,E1 28614.741,E2 28614.741} C_VEL
LIN {X 0,Y 599.976,Z 47.06,A -85,B 0,C 180,E1 28613.428,E2 28613.428} C_VEL
LIN {X 0,Y 598.978,Z 47.191,A -85,B 0,C 180,E1 28612.693,E2 28612.693} C_VEL
LIN {X 0,Y 592.517,Z 47.988,A -85,B 0,C 180,E1 28610.629,E2 28610.629} C_VEL
LIN {X 0,Y 592.003,Z 48.049,A -85,B 0,C 180,E1 28610.092,E2 28610.092} C_VEL
LIN {X 0,Y 592.003,Z 48.052,A -85,B 0,C 180,E1 28606.82,E2 28606.82} C_VEL
LIN {X 0,Y 592.038,Z 48.05,A -85,B 0,C 180,E1 28603.618,E2 28603.618} C_VEL
LIN {X 0,Y 591.991,Z 48.051,A -85,B 0,C 180,E1 28600.462,E2 28600.462} C_VEL
LIN {X 0,Y 592.017,Z 48.051,A -85,B 0,C 180,E1 28597.237,E2 28597.237} C_VEL
LIN {X 0,Y 592.025,Z 48.048,A -85,B 0,C 180,E1 28594.06,E2 28594.06} C_VEL
LIN {X 0,Y 591.985,Z 48.051,A -85,B 0,C 180,E1 28590.831,E2 28590.831} C_VEL
LIN {X 0,Y 592.036,Z 48.054,A -85,B 0,C 180,E1 28587.745,E2 28587.745} C_VEL
LIN {X 0,Y 591.991,Z 48.05,A -85,B 0,C 180,E1 28584.597,E2 28584.597} C_VEL
LIN {X 0,Y 591.989,Z 48.053,A -85,B 0,C 180,E1 28581.287,E2 28581.287} C_VEL
LIN {X 0,Y 592.035,Z 48.051,A -85,B 0,C 180,E1 28578.138,E2 28578.138} C_VEL
LIN {X 0,Y 591.978,Z 48.053,A -85,B 0,C 180,E1 28575.046,E2 28575.046} C_VEL
LIN {X 0,Y 592.017,Z 48.055,A -85,B 0,C 180,E1 28571.857,E2 28571.857} C_VEL
LIN {X 0,Y 591.99,Z 48.053,A -85,B 0,C 180,E1 28568.799,E2 28568.799} C_VEL
LIN {X 0,Y 591.977,Z 48.055,A -85,B 0,C 180,E1 28565.521,E2 28565.521} C_VEL
LIN {X 0,Y 592.052,Z 48.282,A -85,B 0,C 180,E1 28562.596,E2 28562.596} C_VEL
LIN {X 0,Y 592.318,Z 55.545,A -85,B 0,C 180,E1 28561.843,E2 28561.843} C_VEL
LIN {X 0,Y 592.462,Z 87.287,A -85,B 0,C 180,E1 28558.582,E2 28558.582} C_VEL
LIN {X 0,Y 592.334,Z 117.062,A -85,B 0,C 180,E1 28555.433,E2 28555.433} C_VEL
LIN {X 0,Y 592.188,Z 148.276,A -85,B 0,C 180,E1 28552.185,E2 28552.185} C_VEL
LIN {X 0,Y 592.124,Z 175.848,A -85,B 0,C 180,E1 28549.377,E2 28549.377} C_VEL
LIN {X 0,Y 592.316,Z 202.602,A -85,B 0,C 180,E1 28549.034,E2 28549.034} C_VEL
LIN {X 0,Y 592.22,Z 287.638,A -85,B 0,C 180,E1 28547.975,E2 28547.975} C_VEL
LIN {X 0,Y 592.207,Z 302.133,A -85,B 0,C 180,E1 28547.617,E2 28547.617} C_VEL
LIN {X 0,Y 592.166,Z 316.288,A -85,B 0,C 180,E1 28547.084,E2 28547.084} C_VEL
LIN {X 0,Y 592.079,Z 329.845,A -85,B 0,C 180,E1 28546.38,E2 28546.38} C_VEL
LIN {X 0,Y 592.051,Z 342.344,A -85,B 0,C 180,E1 28545.525,E2 28545.525} C_VEL
LIN {X 0,Y 592.008,Z 353.754,A -85,B 0,C 180,E1 28544.524,E2 28544.524} C_VEL
LIN {X 0,Y 591.971,Z 363.19,A -85,B 0,C 180,E1 28543.478,E2 28543.478} C_VEL
LIN {X 0,Y 591.944,Z 371.672,A -85,B 0,C 180,E1 28542.287,E2 28542.287} C_VEL
LIN {X 0,Y 591.927,Z 378.659,A -85,B 0,C 180,E1 28541.003,E2 28541.003} C_VEL
LIN {X 0,Y 591.92,Z 384.129,A -85,B 0,C 180,E1 28539.626,E2 28539.626} C_VEL
LIN {X 0,Y 591.917,Z 387.916,A -85,B 0,C 180,E1 28538.156,E2 28538.156} C_VEL
LIN {X 0,Y 591.916,Z 389.766,A -85,B 0,C 180,E1 28536.661,E2 28536.661} C_VEL
LIN {X 0,Y 591.916,Z 389.755,A -85,B 0,C 180,E1 28535.233,E2 28535.233} C_VEL
LIN {X 0,Y 591.916,Z 387.965,A -85,B 0,C 180,E1 28533.776,E2 28533.776} C_VEL
LIN {X 0,Y 591.918,Z 384.248,A -85,B 0,C 180,E1 28532.323,E2 28532.323} C_VEL
LIN {X 0,Y 591.927,Z 378.943,A -85,B 0,C 180,E1 28530.967,E2 28530.967} C_VEL
LIN {X 0,Y 591.945,Z 372.211,A -85,B 0,C 180,E1 28529.709,E2 28529.709} C_VEL
LIN {X 0,Y 591.97,Z 363.338,A -85,B 0,C 180,E1 28528.451,E2 28528.451} C_VEL
LIN {X 0,Y 592.008,Z 353.752,A -85,B 0,C 180,E1 28527.386,E2 28527.386} C_VEL
LIN {X 0,Y 592.052,Z 342.125,A -85,B 0,C 180,E1 28526.368,E2 28526.368} C_VEL
LIN {X 0,Y 592.079,Z 329.438,A -85,B 0,C 180,E1 28525.505,E2 28525.505} C_VEL
LIN {X 0,Y 592.166,Z 316.078,A -85,B 0,C 180,E1 28524.817,E2 28524.817} C_VEL
LIN {X 0,Y 592.165,Z 301.823,A -85,B 0,C 180,E1 28524.282,E2 28524.282} C_VEL
LIN {X 0,Y 592.178,Z 286.584,A -85,B 0,C 180,E1 28523.914,E2 28523.914} C_VEL
LIN {X 0,Y 592.196,Z 172.307,A -85,B 0,C 180,E1 28522.493,E2 28522.493} C_VEL
LIN {X 0,Y 592.324,Z 123.182,A -85,B 0,C 180,E1 28519.495,E2 28519.495} C_VEL
LIN {X 0,Y 592.569,Z 73.804,A -85,B 0,C 180,E1 28516.435,E2 28516.435} C_VEL
LIN {X 0,Y 592.502,Z 50.051,A -85,B 0,C 180,E1 28514.937,E2 28514.937} C_VEL
LIN {X 0,Y 592.02,Z 48.234,A -85,B 0,C 180,E1 28514.755,E2 28514.755} C_VEL
LIN {X 0,Y 592.025,Z 48.053,A -85,B 0,C 180,E1 28511.691,E2 28511.691} C_VEL
LIN {X 0,Y 592.08,Z 48.368,A -85,B 0,C 180,E1 28511.131,E2 28511.131} C_VEL
LIN {X 0,Y 592.664,Z 51.639,A -85,B 0,C 180,E1 28510.867,E2 28510.867} C_VEL
LIN {X 0,Y 592.453,Z 103.221,A -85,B 0,C 180,E1 28507.645,E2 28507.645} C_VEL
LIN {X 0,Y 592.24,Z 156.193,A -85,B 0,C 180,E1 28504.393,E2 28504.393} C_VEL
LIN {X 0,Y 592.243,Z 172.5,A -85,B 0,C 180,E1 28503.41,E2 28503.41} C_VEL
LIN {X 0,Y 592.228,Z 287.359,A -85,B 0,C 180,E1 28501.979,E2 28501.979} C_VEL
LIN {X 0,Y 592.213,Z 301.992,A -85,B 0,C 180,E1 28501.623,E2 28501.623} C_VEL
LIN {X 0,Y 592.165,Z 316.211,A -85,B 0,C 180,E1 28501.087,E2 28501.087} C_VEL
LIN {X 0,Y 592.086,Z 329.119,A -85,B 0,C 180,E1 28500.423,E2 28500.423} C_VEL
LIN {X 0,Y 592.059,Z 342.262,A -85,B 0,C 180,E1 28499.532,E2 28499.532} C_VEL
LIN {X 0,Y 592.007,Z 354.099,A -85,B 0,C 180,E1 28498.49,E2 28498.49} C_VEL
LIN {X 0,Y 591.969,Z 363.819,A -85,B 0,C 180,E1 28497.398,E2 28497.398} C_VEL
LIN {X 0,Y 591.942,Z 372.171,A -85,B 0,C 180,E1 28496.207,E2 28496.207} C_VEL
LIN {X 0,Y 591.928,Z 379.47,A -85,B 0,C 180,E1 28494.83,E2 28494.83} C_VEL
LIN {X 0,Y 591.919,Z 384.468,A -85,B 0,C 180,E1 28493.516,E2 28493.516} C_VEL
LIN {X 0,Y 591.918,Z 388.1,A -85,B 0,C 180,E1 28492.058,E2 28492.058} C_VEL
LIN {X 0,Y 591.917,Z 389.856,A -85,B 0,C 180,E1 28490.531,E2 28490.531} C_VEL
LIN {X 0,Y 591.916,Z 389.618,A -85,B 0,C 180,E1 28489.032,E2 28489.032} C_VEL
LIN {X 0,Y 591.917,Z 387.65,A -85,B 0,C 180,E1 28487.624,E2 28487.624} C_VEL
LIN {X 0,Y 591.92,Z 383.729,A -85,B 0,C 180,E1 28486.161,E2 28486.161} C_VEL
LIN {X 0,Y 591.93,Z 378.052,A -85,B 0,C 180,E1 28484.78,E2 28484.78} C_VEL
LIN {X 0,Y 591.946,Z 370.95,A -85,B 0,C 180,E1 28483.511,E2 28483.511} C_VEL
LIN {X 0,Y 591.976,Z 362.018,A -85,B 0,C 180,E1 28482.286,E2 28482.286} C_VEL
LIN {X 0,Y 592.018,Z 351.076,A -85,B 0,C 180,E1 28481.127,E2 28481.127} C_VEL
LIN {X 0,Y 592.058,Z 338.973,A -85,B 0,C 180,E1 28480.133,E2 28480.133} C_VEL
LIN {X 0,Y 592.118,Z 326.554,A -85,B 0,C 180,E1 28479.341,E2 28479.341} C_VEL
LIN {X 0,Y 592.18,Z 312.482,A -85,B 0,C 180,E1 28478.662,E2 28478.662} C_VEL
LIN {X 0,Y 592.223,Z 296.996,A -85,B 0,C 180,E1 28478.144,E2 28478.144} C_VEL
LIN {X 0,Y 592.25,Z 281.762,A -85,B 0,C 180,E1 28477.841,E2 28477.841} C_VEL
LIN {X 0,Y 592.151,Z 176.009,A -85,B 0,C 180,E1 28476.538,E2 28476.538} C_VEL
LIN {X 0,Y 592.232,Z 145.962,A -85,B 0,C 180,E1 28473.487,E2 28473.487} C_VEL
LIN {X 0,Y 592.351,Z 114.424,A -85,B 0,C 180,E1 28470.2,E2 28470.2} C_VEL
LIN {X 0,Y 592.523,Z 85.445,A -85,B 0,C 180,E1 28467.105,E2 28467.105} C_VEL
LIN {X 0,Y 592.837,Z 56.662,A -85,B 0,C 180,E1 28463.92,E2 28463.92} C_VEL
LIN {X 0,Y 592.66,Z 50.727,A -85,B 0,C 180,E1 28463.252,E2 28463.252} C_VEL
LIN {X 0,Y 592.001,Z 48.143,A -85,B 0,C 180,E1 28462.885,E2 28462.885} C_VEL
LIN {X 0,Y 592.035,Z 48.055,A -85,B 0,C 180,E1 28459.741,E2 28459.741} C_VEL
LIN {X 0,Y 592.003,Z 48.051,A -85,B 0,C 180,E1 28456.585,E2 28456.585} C_VEL
LIN {X 0,Y 591.992,Z 48.054,A -85,B 0,C 180,E1 28453.379,E2 28453.379} C_VEL
LIN {X 0,Y 592.039,Z 48.051,A -85,B 0,C 180,E1 28450.214,E2 28450.214} C_VEL
LIN {X 0,Y 591.983,Z 48.052,A -85,B 0,C 180,E1 28447.083,E2 28447.083} C_VEL
LIN {X 0,Y 592.01,Z 48.055,A -85,B 0,C 180,E1 28443.874,E2 28443.874} C_VEL
LIN {X 0,Y 592.006,Z 48.051,A -85,B 0,C 180,E1 28440.774,E2 28440.774} C_VEL
LIN {X 0,Y 591.978,Z 48.054,A -85,B 0,C 180,E1 28437.58,E2 28437.58} C_VEL
LIN {X 0,Y 592.041,Z 48.053,A -85,B 0,C 180,E1 28434.476,E2 28434.476} C_VEL
LIN {X 0,Y 591.975,Z 48.053,A -85,B 0,C 180,E1 28431.355,E2 28431.355} C_VEL
LIN {X 0,Y 591.994,Z 48.055,A -85,B 0,C 180,E1 28428.109,E2 28428.109} C_VEL
LIN {X 0,Y 591.994,Z 48.052,A -85,B 0,C 180,E1 28425.124,E2 28425.124} C_VEL
LIN {X 0,Y 591.97,Z 48.054,A -85,B 0,C 180,E1 28421.894,E2 28421.894} C_VEL
LIN {X 0,Y 592.037,Z 48.054,A -85,B 0,C 180,E1 28418.787,E2 28418.787} C_VEL
LIN {X 0,Y 591.964,Z 48.054,A -85,B 0,C 180,E1 28415.768,E2 28415.768} C_VEL
LIN {X 0,Y 592.011,Z 48.055,A -85,B 0,C 180,E1 28412.653,E2 28412.653} C_VEL
LIN {X 0,Y 591.968,Z 48.055,A -85,B 0,C 180,E1 28409.666,E2 28409.666} C_VEL
LIN {X 0,Y 591.967,Z 48.055,A -85,B 0,C 180,E1 28406.358,E2 28406.358} C_VEL
LIN {X 0,Y 591.998,Z 48.055,A -85,B 0,C 180,E1 28403.402,E2 28403.402} C_VEL
LIN {X 0,Y 591.957,Z 48.056,A -85,B 0,C 180,E1 28400.322,E2 28400.322} C_VEL
LIN {X 0,Y 592.028,Z 48.056,A -85,B 0,C 180,E1 28397.278,E2 28397.278} C_VEL
LIN {X 0,Y 591.957,Z 48.056,A -85,B 0,C 180,E1 28394.234,E2 28394.234} C_VEL
LIN {X 0,Y 592.004,Z 48.055,A -85,B 0,C 180,E1 28391.071,E2 28391.071} C_VEL
LIN {X 0,Y 591.964,Z 48.056,A -85,B 0,C 180,E1 28388.184,E2 28388.184} C_VEL
LIN {X 0,Y 591.981,Z 48.056,A -85,B 0,C 180,E1 28384.93,E2 28384.93} C_VEL
LIN {X 0,Y 591.986,Z 48.056,A -85,B 0,C 180,E1 28382.019,E2 28382.019} C_VEL
LIN {X 0,Y 591.999,Z 48.3,A -85,B 0,C 180,E1 28380.472,E2 28380.472} C_VEL
LIN {X 0,Y 593.247,Z 53,A -85,B 0,C 180,E1 28380.038,E2 28380.038} C_VEL
LIN {X 0,Y 593.12,Z 96.992,A -85,B 0,C 180,E1 28377.021,E2 28377.021} C_VEL
LIN {X 0,Y 592.849,Z 145.038,A -85,B 0,C 180,E1 28373.771,E2 28373.771} C_VEL
LIN {X 0,Y 592.863,Z 158.178,A -85,B 0,C 180,E1 28372.925,E2 28372.925} C_VEL
LIN {X 0,Y 593.101,Z 171.968,A -85,B 0,C 180,E1 28372.735,E2 28372.735} C_VEL
LIN {X 0,Y 592.851,Z 367.301,A -85,B 0,C 180,E1 28370.227,E2 28370.227} C_VEL
LIN {X 0,Y 592.771,Z 386.296,A -85,B 0,C 180,E1 28369.797,E2 28369.797} C_VEL
LIN {X 0,Y 592.675,Z 404.393,A -85,B 0,C 180,E1 28369.207,E2 28369.207} C_VEL
LIN {X 0,Y 592.565,Z 422.04,A -85,B 0,C 180,E1 28368.444,E2 28368.444} C_VEL
LIN {X 0,Y 592.459,Z 438.691,A -85,B 0,C 180,E1 28367.538,E2 28367.538} C_VEL
LIN {X 0,Y 592.341,Z 454.63,A -85,B 0,C 180,E1 28366.474,E2 28366.474} C_VEL
LIN {X 0,Y 592.23,Z 469.556,A -85,B 0,C 180,E1 28365.271,E2 28365.271} C_VEL
LIN {X 0,Y 592.136,Z 483.015,A -85,B 0,C 180,E1 28363.974,E2 28363.974} C_VEL
LIN {X 0,Y 592.056,Z 495.422,A -85,B 0,C 180,E1 28362.546,E2 28362.546} C_VEL
LIN {X 0,Y 592,Z 506.585,A -85,B 0,C 180,E1 28361.003,E2 28361.003} C_VEL
LIN {X 0,Y 591.955,Z 516.472,A -85,B 0,C 180,E1 28359.332,E2 28359.332} C_VEL
LIN {X 0,Y 591.935,Z 524.771,A -85,B 0,C 180,E1 28357.571,E2 28357.571} C_VEL
LIN {X 0,Y 591.918,Z 531.25,A -85,B 0,C 180,E1 28355.772,E2 28355.772} C_VEL
LIN {X 0,Y 591.915,Z 535.873,A -85,B 0,C 180,E1 28353.972,E2 28353.972} C_VEL
LIN {X 0,Y 591.913,Z 538.788,A -85,B 0,C 180,E1 28352.13,E2 28352.13} C_VEL
LIN {X 0,Y 591.907,Z 539.939,A -85,B 0,C 180,E1 28350.291,E2 28350.291} C_VEL
LIN {X 0,Y 591.914,Z 539.35,A -85,B 0,C 180,E1 28348.452,E2 28348.452} C_VEL
LIN {X 0,Y 591.907,Z 537.008,A -85,B 0,C 180,E1 28346.611,E2 28346.611} C_VEL
LIN {X 0,Y 591.919,Z 533.1,A -85,B 0,C 180,E1 28344.864,E2 28344.864} C_VEL
LIN {X 0,Y 591.93,Z 527.47,A -85,B 0,C 180,E1 28343.113,E2 28343.113} C_VEL
LIN {X 0,Y 591.943,Z 520.428,A -85,B 0,C 180,E1 28341.453,E2 28341.453} C_VEL
LIN {X 0,Y 591.977,Z 511.517,A -85,B 0,C 180,E1 28339.786,E2 28339.786} C_VEL
LIN {X 0,Y 592.024,Z 501.154,A -85,B 0,C 180,E1 28338.209,E2 28338.209} C_VEL
LIN {X 0,Y 592.094,Z 489.356,A -85,B 0,C 180,E1 28336.724,E2 28336.724} C_VEL
LIN {X 0,Y 592.192,Z 475.589,A -85,B 0,C 180,E1 28335.28,E2 28335.28} C_VEL
LIN {X 0,Y 592.306,Z 460.611,A -85,B 0,C 180,E1 28333.979,E2 28333.979} C_VEL
LIN {X 0,Y 592.422,Z 444.44,A -85,B 0,C 180,E1 28332.822,E2 28332.822} C_VEL
LIN {X 0,Y 592.535,Z 428.063,A -85,B 0,C 180,E1 28331.862,E2 28331.862} C_VEL
LIN {X 0,Y 592.649,Z 411.154,A -85,B 0,C 180,E1 28331.063,E2 28331.063} C_VEL
LIN {X 0,Y 592.752,Z 392.874,A -85,B 0,C 180,E1 28330.397,E2 28330.397} C_VEL
LIN {X 0,Y 592.831,Z 374.359,A -85,B 0,C 180,E1 28329.912,E2 28329.912} C_VEL
LIN {X 0,Y 592.88,Z 354.558,A -85,B 0,C 180,E1 28329.587,E2 28329.587} C_VEL
LIN {X 0,Y 593,Z 155.102,A -85,B 0,C 180,E1 28327.038,E2 28327.038} C_VEL
LIN {X 0,Y 593.308,Z 75.967,A -85,B 0,C 180,E1 28323.88,E2 28323.88} C_VEL
LIN {X 0,Y 593.183,Z 51.428,A -85,B 0,C 180,E1 28322.872,E2 28322.872} C_VEL
LIN {X 0,Y 592.09,Z 48.462,A -85,B 0,C 180,E1 28322.654,E2 28322.654} C_VEL
LIN {X 0,Y 592.027,Z 48.054,A -85,B 0,C 180,E1 28322.218,E2 28322.218} C_VEL
LIN {X 0,Y 592.019,Z 48.05,A -85,B 0,C 180,E1 28318.996,E2 28318.996} C_VEL
LIN {X 0,Y 592.031,Z 48.053,A -85,B 0,C 180,E1 28315.78,E2 28315.78} C_VEL
LIN {X 0,Y 592.03,Z 48.047,A -85,B 0,C 180,E1 28312.435,E2 28312.435} C_VEL
LIN {X 0,Y 592.017,Z 48.051,A -85,B 0,C 180,E1 28309.316,E2 28309.316} C_VEL
LIN {X 0,Y 592.027,Z 48.052,A -85,B 0,C 180,E1 28306.149,E2 28306.149} C_VEL
LIN {X 0,Y 592.034,Z 48.046,A -85,B 0,C 180,E1 28302.867,E2 28302.867} C_VEL
LIN {X 0,Y 592.017,Z 48.052,A -85,B 0,C 180,E1 28299.636,E2 28299.636} C_VEL
LIN {X 0,Y 592.028,Z 48.05,A -85,B 0,C 180,E1 28296.476,E2 28296.476} C_VEL
LIN {X 0,Y 592.018,Z 48.048,A -85,B 0,C 180,E1 28293.282,E2 28293.282} C_VEL
LIN {X 0,Y 592.02,Z 48.053,A -85,B 0,C 180,E1 28289.96,E2 28289.96} C_VEL
LIN {X 0,Y 592.031,Z 48.048,A -85,B 0,C 180,E1 28286.803,E2 28286.803} C_VEL
LIN {X 0,Y 592.008,Z 48.048,A -85,B 0,C 180,E1 28283.595,E2 28283.595} C_VEL
LIN {X 0,Y 592.032,Z 48.054,A -85,B 0,C 180,E1 28280.359,E2 28280.359} C_VEL
LIN {X 0,Y 592.037,Z 48.047,A -85,B 0,C 180,E1 28277.088,E2 28277.088} C_VEL
LIN {X 0,Y 592.004,Z 48.049,A -85,B 0,C 180,E1 28273.876,E2 28273.876} C_VEL
LIN {X 0,Y 592.032,Z 48.054,A -85,B 0,C 180,E1 28270.608,E2 28270.608} C_VEL
LIN {X 0,Y 592.034,Z 48.047,A -85,B 0,C 180,E1 28267.374,E2 28267.374} C_VEL
LIN {X 0,Y 592,Z 48.05,A -85,B 0,C 180,E1 28264.165,E2 28264.165} C_VEL
LIN {X 0,Y 592.039,Z 48.054,A -85,B 0,C 180,E1 28260.967,E2 28260.967} C_VEL
LIN {X 0,Y 592.025,Z 48.047,A -85,B 0,C 180,E1 28257.677,E2 28257.677} C_VEL
LIN {X 0,Y 591.998,Z 48.052,A -85,B 0,C 180,E1 28254.475,E2 28254.475} C_VEL
LIN {X 0,Y 592.036,Z 48.051,A -85,B 0,C 180,E1 28251.355,E2 28251.355} C_VEL
LIN {X 0,Y 592.003,Z 48.049,A -85,B 0,C 180,E1 28250.092,E2 28250.092} C_VEL
LIN {X 0,Y 591.043,Z 48.176,A -85,B 0,C 180,E1 28249.346,E2 28249.346} C_VEL
LIN {X 0,Y 584.513,Z 48.992,A -85,B 0,C 180,E1 28247.2,E2 28247.2} C_VEL
LIN {X 0,Y 584.058,Z 49.04,A -85,B 0,C 180,E1 28246.709,E2 28246.709} C_VEL
LIN {X 0,Y 584.099,Z 49.041,A -85,B 0,C 180,E1 28243.491,E2 28243.491} C_VEL
LIN {X 0,Y 584.059,Z 49.039,A -85,B 0,C 180,E1 28240.29,E2 28240.29} C_VEL
LIN {X 0,Y 584.055,Z 49.038,A -85,B 0,C 180,E1 28236.919,E2 28236.919} C_VEL
LIN {X 0,Y 584.1,Z 49.039,A -85,B 0,C 180,E1 28233.76,E2 28233.76} C_VEL
LIN {X 0,Y 584.05,Z 49.038,A -85,B 0,C 180,E1 28230.572,E2 28230.572} C_VEL
LIN {X 0,Y 584.058,Z 49.043,A -85,B 0,C 180,E1 28227.25,E2 28227.25} C_VEL
LIN {X 0,Y 584.097,Z 49.038,A -85,B 0,C 180,E1 28224.062,E2 28224.062} C_VEL
LIN {X 0,Y 584.042,Z 49.041,A -85,B 0,C 180,E1 28220.949,E2 28220.949} C_VEL
LIN {X 0,Y 584.079,Z 49.044,A -85,B 0,C 180,E1 28217.719,E2 28217.719} C_VEL
LIN {X 0,Y 584.054,Z 49.041,A -85,B 0,C 180,E1 28214.715,E2 28214.715} C_VEL
LIN {X 0,Y 584.041,Z 49.043,A -85,B 0,C 180,E1 28211.423,E2 28211.423} C_VEL
LIN {X 0,Y 584.097,Z 49.043,A -85,B 0,C 180,E1 28208.29,E2 28208.29} C_VEL
LIN {X 0,Y 584.035,Z 49.044,A -85,B 0,C 180,E1 28205.234,E2 28205.234} C_VEL
LIN {X 0,Y 584.103,Z 49.316,A -85,B 0,C 180,E1 28202.745,E2 28202.745} C_VEL
LIN {X 0,Y 584.509,Z 53.251,A -85,B 0,C 180,E1 28202.324,E2 28202.324} C_VEL
LIN {X 0,Y 584.687,Z 83.63,A -85,B 0,C 180,E1 28199.223,E2 28199.223} C_VEL
LIN {X 0,Y 584.601,Z 112.552,A -85,B 0,C 180,E1 28196.183,E2 28196.183} C_VEL
LIN {X 0,Y 584.408,Z 144.038,A -85,B 0,C 180,E1 28192.852,E2 28192.852} C_VEL
LIN {X 0,Y 584.206,Z 175.491,A -85,B 0,C 180,E1 28189.585,E2 28189.585} C_VEL
LIN {X 0,Y 584.545,Z 180.922,A -85,B 0,C 180,E1 28189.48,E2 28189.48} C_VEL
LIN {X 0,Y 584.392,Z 287.666,A -85,B 0,C 180,E1 28188.139,E2 28188.139} C_VEL
LIN {X 0,Y 584.363,Z 301.933,A -85,B 0,C 180,E1 28187.782,E2 28187.782} C_VEL
LIN {X 0,Y 584.296,Z 315.992,A -85,B 0,C 180,E1 28187.25,E2 28187.25} C_VEL
LIN {X 0,Y 584.192,Z 329.023,A -85,B 0,C 180,E1 28186.572,E2 28186.572} C_VEL
LIN {X 0,Y 584.122,Z 341.898,A -85,B 0,C 180,E1 28185.69,E2 28185.69} C_VEL
LIN {X 0,Y 584.057,Z 353.413,A -85,B 0,C 180,E1 28184.676,E2 28184.676} C_VEL
LIN {X 0,Y 583.999,Z 363.325,A -85,B 0,C 180,E1 28183.564,E2 28183.564} C_VEL
LIN {X 0,Y 583.959,Z 371.773,A -85,B 0,C 180,E1 28182.357,E2 28182.357} C_VEL
LIN {X 0,Y 583.933,Z 378.74,A -85,B 0,C 180,E1 28181.055,E2 28181.055} C_VEL
LIN {X 0,Y 583.922,Z 384.182,A -85,B 0,C 180,E1 28179.659,E2 28179.659} C_VEL
LIN {X 0,Y 583.918,Z 387.949,A -85,B 0,C 180,E1 28178.17,E2 28178.17} C_VEL
LIN {X 0,Y 583.916,Z 389.756,A -85,B 0,C 180,E1 28176.686,E2 28176.686} C_VEL
LIN {X 0,Y 583.916,Z 389.811,A -85,B 0,C 180,E1 28175.305,E2 28175.305} C_VEL
LIN {X 0,Y 583.917,Z 388.11,A -85,B 0,C 180,E1 28173.828,E2 28173.828} C_VEL
LIN {X 0,Y 583.919,Z 384.499,A -85,B 0,C 180,E1 28172.354,E2 28172.354} C_VEL
LIN {X 0,Y 583.933,Z 379.315,A -85,B 0,C 180,E1 28170.98,E2 28170.98} C_VEL
LIN {X 0,Y 583.959,Z 372.113,A -85,B 0,C 180,E1 28169.607,E2 28169.607} C_VEL
LIN {X 0,Y 584,Z 363.215,A -85,B 0,C 180,E1 28168.331,E2 28168.331} C_VEL
LIN {X 0,Y 584.056,Z 353.587,A -85,B 0,C 180,E1 28167.252,E2 28167.252} C_VEL
LIN {X 0,Y 584.121,Z 342.545,A -85,B 0,C 180,E1 28166.27,E2 28166.27} C_VEL
LIN {X 0,Y 584.179,Z 329.811,A -85,B 0,C 180,E1 28165.385,E2 28165.385} C_VEL
LIN {X 0,Y 584.297,Z 315.718,A -85,B 0,C 180,E1 28164.648,E2 28164.648} C_VEL
LIN {X 0,Y 584.322,Z 301.284,A -85,B 0,C 180,E1 28164.106,E2 28164.106} C_VEL
LIN {X 0,Y 584.35,Z 286.141,A -85,B 0,C 180,E1 28163.743,E2 28163.743} C_VEL
LIN {X 0,Y 584.355,Z 172.241,A -85,B 0,C 180,E1 28162.305,E2 28162.305} C_VEL
LIN {X 0,Y 584.571,Z 123.575,A -85,B 0,C 180,E1 28159.295,E2 28159.295} C_VEL
LIN {X 0,Y 584.915,Z 73.556,A -85,B 0,C 180,E1 28156.153,E2 28156.153} C_VEL
LIN {X 0,Y 585.019,Z 52.749,A -85,B 0,C 180,E1 28154.841,E2 28154.841} C_VEL
LIN {X 0,Y 584.092,Z 49.324,A -85,B 0,C 180,E1 28154.571,E2 28154.571} C_VEL
LIN {X 0,Y 584.077,Z 49.043,A -85,B 0,C 180,E1 28152.79,E2 28152.79} C_VEL
LIN {X 0,Y 584.132,Z 49.298,A -85,B 0,C 180,E1 28151.409,E2 28151.409} C_VEL
LIN {X 0,Y 585.09,Z 53.439,A -85,B 0,C 180,E1 28151.053,E2 28151.053} C_VEL
LIN {X 0,Y 584.73,Z 104.186,A -85,B 0,C 180,E1 28147.826,E2 28147.826} C_VEL
LIN {X 0,Y 584.428,Z 156.532,A -85,B 0,C 180,E1 28144.569,E2 28144.569} C_VEL
LIN {X 0,Y 584.44,Z 172.925,A -85,B 0,C 180,E1 28143.585,E2 28143.585} C_VEL
LIN {X 0,Y 584.4,Z 287.525,A -85,B 0,C 180,E1 28142.14,E2 28142.14} C_VEL
LIN {X 0,Y 584.364,Z 302.533,A -85,B 0,C 180,E1 28141.764,E2 28141.764} C_VEL
LIN {X 0,Y 584.29,Z 317.477,A -85,B 0,C 180,E1 28141.183,E2 28141.183} C_VEL
LIN {X 0,Y 584.176,Z 330.742,A -85,B 0,C 180,E1 28140.466,E2 28140.466} C_VEL
LIN {X 0,Y 584.128,Z 342.77,A -85,B 0,C 180,E1 28139.622,E2 28139.622} C_VEL
LIN {X 0,Y 584.052,Z 354.626,A -85,B 0,C 180,E1 28138.555,E2 28138.555} C_VEL
LIN {X 0,Y 583.992,Z 364.887,A -85,B 0,C 180,E1 28137.363,E2 28137.363} C_VEL
LIN {X 0,Y 583.953,Z 373.041,A -85,B 0,C 180,E1 28136.143,E2 28136.143} C_VEL
LIN {X 0,Y 583.933,Z 379.561,A -85,B 0,C 180,E1 28134.877,E2 28134.877} C_VEL
LIN {X 0,Y 583.92,Z 384.901,A -85,B 0,C 180,E1 28133.424,E2 28133.424} C_VEL
LIN {X 0,Y 583.918,Z 388.129,A -85,B 0,C 180,E1 28132.068,E2 28132.068} C_VEL
LIN {X 0,Y 583.917,Z 389.844,A -85,B 0,C 180,E1 28130.558,E2 28130.558} C_VEL
LIN {X 0,Y 583.916,Z 389.63,A -85,B 0,C 180,E1 28129.038,E2 28129.038} C_VEL
LIN {X 0,Y 583.917,Z 387.884,A -85,B 0,C 180,E1 28127.705,E2 28127.705} C_VEL
LIN {X 0,Y 583.922,Z 384.111,A -85,B 0,C 180,E1 28126.229,E2 28126.229} C_VEL
LIN {X 0,Y 583.935,Z 378.738,A -85,B 0,C 180,E1 28124.856,E2 28124.856} C_VEL
LIN {X 0,Y 583.96,Z 372.025,A -85,B 0,C 180,E1 28123.592,E2 28123.592} C_VEL
LIN {X 0,Y 584.001,Z 362.966,A -85,B 0,C 180,E1 28122.301,E2 28122.301} C_VEL
LIN {X 0,Y 584.057,Z 353.366,A -85,B 0,C 180,E1 28121.231,E2 28121.231} C_VEL
LIN {X 0,Y 584.127,Z 342.088,A -85,B 0,C 180,E1 28120.233,E2 28120.233} C_VEL
LIN {X 0,Y 584.215,Z 328.776,A -85,B 0,C 180,E1 28119.324,E2 28119.324} C_VEL
LIN {X 0,Y 584.295,Z 315.434,A -85,B 0,C 180,E1 28118.637,E2 28118.637} C_VEL
LIN {X 0,Y 584.369,Z 301.228,A -85,B 0,C 180,E1 28118.106,E2 28118.106} C_VEL
LIN {X 0,Y 584.419,Z 285.597,A -85,B 0,C 180,E1 28117.734,E2 28117.734} C_VEL
LIN {X 0,Y 584.325,Z 176.596,A -85,B 0,C 180,E1 28116.369,E2 28116.369} C_VEL
LIN {X 0,Y 584.224,Z 175.072,A -85,B 0,C 180,E1 28116.285,E2 28116.285} C_VEL
LIN {X 0,Y 584.376,Z 143.785,A -85,B 0,C 180,E1 28113.03,E2 28113.03} C_VEL
LIN {X 0,Y 584.614,Z 113.722,A -85,B 0,C 180,E1 28109.848,E2 28109.848} C_VEL
LIN {X 0,Y 584.968,Z 83.171,A -85,B 0,C 180,E1 28106.495,E2 28106.495} C_VEL
LIN {X 0,Y 585.308,Z 55.568,A -85,B 0,C 180,E1 28103.402,E2 28103.402} C_VEL
LIN {X 0,Y 584.947,Z 52.568,A -85,B 0,C 180,E1 28103.044,E2 28103.044} C_VEL
LIN {X 0,Y 584.071,Z 49.111,A -85,B 0,C 180,E1 28102.549,E2 28102.549} C_VEL
LIN {X 0,Y 584.054,Z 49.044,A -85,B 0,C 180,E1 28099.19,E2 28099.19} C_VEL
LIN {X 0,Y 584.101,Z 49.042,A -85,B 0,C 180,E1 28095.998,E2 28095.998} C_VEL
LIN {X 0,Y 584.051,Z 49.041,A -85,B 0,C 180,E1 28092.859,E2 28092.859} C_VEL
LIN {X 0,Y 584.057,Z 49.042,A -85,B 0,C 180,E1 28089.559,E2 28089.559} C_VEL
LIN {X 0,Y 584.095,Z 49.04,A -85,B 0,C 180,E1 28086.389,E2 28086.389} C_VEL
LIN {X 0,Y 584.042,Z 49.042,A -85,B 0,C 180,E1 28083.239,E2 28083.239} C_VEL
LIN {X 0,Y 584.086,Z 49.044,A -85,B 0,C 180,E1 28080.098,E2 28080.098} C_VEL
LIN {X 0,Y 584.055,Z 49.041,A -85,B 0,C 180,E1 28076.958,E2 28076.958} C_VEL
LIN {X 0,Y 584.04,Z 49.043,A -85,B 0,C 180,E1 28073.71,E2 28073.71} C_VEL
LIN {X 0,Y 584.096,Z 49.041,A -85,B 0,C 180,E1 28070.641,E2 28070.641} C_VEL
LIN {X 0,Y 584.032,Z 49.043,A -85,B 0,C 180,E1 28067.543,E2 28067.543} C_VEL
LIN {X 0,Y 584.077,Z 49.044,A -85,B 0,C 180,E1 28064.41,E2 28064.41} C_VEL
LIN {X 0,Y 584.043,Z 49.042,A -85,B 0,C 180,E1 28061.329,E2 28061.329} C_VEL
LIN {X 0,Y 584.035,Z 49.043,A -85,B 0,C 180,E1 28058.086,E2 28058.086} C_VEL
LIN {X 0,Y 584.075,Z 49.043,A -85,B 0,C 180,E1 28055.095,E2 28055.095} C_VEL
LIN {X 0,Y 584.025,Z 49.044,A -85,B 0,C 180,E1 28052.025,E2 28052.025} C_VEL
LIN {X 0,Y 584.094,Z 49.044,A -85,B 0,C 180,E1 28048.986,E2 28048.986} C_VEL
LIN {X 0,Y 584.024,Z 49.044,A -85,B 0,C 180,E1 28045.838,E2 28045.838} C_VEL
LIN {X 0,Y 584.036,Z 49.045,A -85,B 0,C 180,E1 28042.573,E2 28042.573} C_VEL
LIN {X 0,Y 584.049,Z 49.045,A -85,B 0,C 180,E1 28039.547,E2 28039.547} C_VEL
LIN {X 0,Y 584.018,Z 49.044,A -85,B 0,C 180,E1 28036.374,E2 28036.374} C_VEL
LIN {X 0,Y 584.09,Z 49.044,A -85,B 0,C 180,E1 28033.321,E2 28033.321} C_VEL
LIN {X 0,Y 584.022,Z 49.045,A -85,B 0,C 180,E1 28030.198,E2 28030.198} C_VEL
LIN {X 0,Y 584.057,Z 49.044,A -85,B 0,C 180,E1 28027.056,E2 28027.056} C_VEL
LIN {X 0,Y 584.04,Z 49.046,A -85,B 0,C 180,E1 28024.043,E2 28024.043} C_VEL
LIN {X 0,Y 584.058,Z 49.226,A -85,B 0,C 180,E1 28020.838,E2 28020.838} C_VEL
LIN {X 0,Y 585.895,Z 55.699,A -85,B 0,C 180,E1 28020.228,E2 28020.228} C_VEL
LIN {X 0,Y 585.684,Z 99.558,A -85,B 0,C 180,E1 28017.198,E2 28017.198} C_VEL
LIN {X 0,Y 585.33,Z 146.613,A -85,B 0,C 180,E1 28013.989,E2 28013.989} C_VEL
LIN {X 0,Y 585.313,Z 158.079,A -85,B 0,C 180,E1 28013.24,E2 28013.24} C_VEL
LIN {X 0,Y 585.733,Z 163.874,A -85,B 0,C 180,E1 28013.143,E2 28013.143} C_VEL
LIN {X 0,Y 585.341,Z 367.301,A -85,B 0,C 180,E1 28010.498,E2 28010.498} C_VEL
LIN {X 0,Y 585.222,Z 386.295,A -85,B 0,C 180,E1 28010.064,E2 28010.064} C_VEL
LIN {X 0,Y 585.079,Z 404.39,A -85,B 0,C 180,E1 28009.466,E2 28009.466} C_VEL
LIN {X 0,Y 584.915,Z 421.935,A -85,B 0,C 180,E1 28008.7,E2 28008.7} C_VEL
LIN {X 0,Y 584.738,Z 439.211,A -85,B 0,C 180,E1 28007.744,E2 28007.744} C_VEL
LIN {X 0,Y 584.559,Z 455.227,A -85,B 0,C 180,E1 28006.654,E2 28006.654} C_VEL
LIN {X 0,Y 584.393,Z 470.094,A -85,B 0,C 180,E1 28005.431,E2 28005.431} C_VEL
LIN {X 0,Y 584.245,Z 483.941,A -85,B 0,C 180,E1 28004.065,E2 28004.065} C_VEL
LIN {X 0,Y 584.125,Z 496.682,A -85,B 0,C 180,E1 28002.556,E2 28002.556} C_VEL
LIN {X 0,Y 584.042,Z 507.864,A -85,B 0,C 180,E1 28000.955,E2 28000.955} C_VEL
LIN {X 0,Y 583.976,Z 517.507,A -85,B 0,C 180,E1 27999.262,E2 27999.262} C_VEL
LIN {X 0,Y 583.943,Z 525.402,A -85,B 0,C 180,E1 27997.522,E2 27997.522} C_VEL
LIN {X 0,Y 583.922,Z 531.41,A -85,B 0,C 180,E1 27995.799,E2 27995.799} C_VEL
LIN {X 0,Y 583.914,Z 535.873,A -85,B 0,C 180,E1 27994.026,E2 27994.026} C_VEL
LIN {X 0,Y 583.913,Z 538.789,A -85,B 0,C 180,E1 27992.16,E2 27992.16} C_VEL
LIN {X 0,Y 583.907,Z 539.939,A -85,B 0,C 180,E1 27990.295,E2 27990.295} C_VEL
LIN {X 0,Y 583.913,Z 539.349,A -85,B 0,C 180,E1 27988.431,E2 27988.431} C_VEL
LIN {X 0,Y 583.907,Z 537.007,A -85,B 0,C 180,E1 27986.565,E2 27986.565} C_VEL
LIN {X 0,Y 583.922,Z 533.1,A -85,B 0,C 180,E1 27984.794,E2 27984.794} C_VEL
LIN {X 0,Y 583.935,Z 527.47,A -85,B 0,C 180,E1 27983.018,E2 27983.018} C_VEL
LIN {X 0,Y 583.96,Z 520.429,A -85,B 0,C 180,E1 27981.335,E2 27981.335} C_VEL
LIN {X 0,Y 584.015,Z 511.518,A -85,B 0,C 180,E1 27979.645,E2 27979.645} C_VEL
LIN {X 0,Y 584.086,Z 501.155,A -85,B 0,C 180,E1 27978.047,E2 27978.047} C_VEL
LIN {X 0,Y 584.195,Z 489.357,A -85,B 0,C 180,E1 27976.541,E2 27976.541} C_VEL
LIN {X 0,Y 584.343,Z 475.588,A -85,B 0,C 180,E1 27975.078,E2 27975.078} C_VEL
LIN {X 0,Y 584.508,Z 460.613,A -85,B 0,C 180,E1 27973.76,E2 27973.76} C_VEL
LIN {X 0,Y 584.686,Z 444.444,A -85,B 0,C 180,E1 27972.588,E2 27972.588} C_VEL
LIN {X 0,Y 584.866,Z 427.51,A -85,B 0,C 180,E1 27971.586,E2 27971.586} C_VEL
LIN {X 0,Y 585.033,Z 410.833,A -85,B 0,C 180,E1 27970.793,E2 27970.793} C_VEL
LIN {X 0,Y 585.188,Z 392.666,A -85,B 0,C 180,E1 27970.127,E2 27970.127} C_VEL
LIN {X 0,Y 585.309,Z 374.196,A -85,B 0,C 180,E1 27969.639,E2 27969.639} C_VEL
LIN {X 0,Y 585.382,Z 354.294,A -85,B 0,C 180,E1 27969.31,E2 27969.31} C_VEL
LIN {X 0,Y 585.609,Z 155.82,A -85,B 0,C 180,E1 27966.746,E2 27966.746} C_VEL
LIN {X 0,Y 586,Z 81.253,A -85,B 0,C 180,E1 27963.748,E2 27963.748} C_VEL
LIN {X 0,Y 585.925,Z 54.364,A -85,B 0,C 180,E1 27962.65,E2 27962.65} C_VEL
LIN {X 0,Y 584.166,Z 49.51,A -85,B 0,C 180,E1 27962.338,E2 27962.338} C_VEL
LIN {X 0,Y 584.086,Z 49.04,A -85,B 0,C 180,E1 27962.14,E2 27962.14} C_VEL
LIN {X 0,Y 584.081,Z 49.039,A -85,B 0,C 180,E1 27958.986,E2 27958.986} C_VEL
LIN {X 0,Y 584.095,Z 49.042,A -85,B 0,C 180,E1 27955.725,E2 27955.725} C_VEL
LIN {X 0,Y 584.091,Z 49.037,A -85,B 0,C 180,E1 27952.426,E2 27952.426} C_VEL
LIN {X 0,Y 584.077,Z 49.039,A -85,B 0,C 180,E1 27949.163,E2 27949.163} C_VEL
LIN {X 0,Y 584.096,Z 49.043,A -85,B 0,C 180,E1 27945.968,E2 27945.968} C_VEL
LIN {X 0,Y 584.093,Z 49.036,A -85,B 0,C 180,E1 27942.604,E2 27942.604} C_VEL
LIN {X 0,Y 584.074,Z 49.039,A -85,B 0,C 180,E1 27939.428,E2 27939.428} C_VEL
LIN {X 0,Y 584.095,Z 49.043,A -85,B 0,C 180,E1 27936.198,E2 27936.198} C_VEL
LIN {X 0,Y 584.096,Z 49.035,A -85,B 0,C 180,E1 27932.864,E2 27932.864} C_VEL
LIN {X 0,Y 584.071,Z 49.039,A -85,B 0,C 180,E1 27929.587,E2 27929.587} C_VEL
LIN {X 0,Y 584.097,Z 49.044,A -85,B 0,C 180,E1 27926.318,E2 27926.318} C_VEL
LIN {X 0,Y 584.096,Z 49.035,A -85,B 0,C 180,E1 27922.972,E2 27922.972} C_VEL
LIN {X 0,Y 584.065,Z 49.039,A -85,B 0,C 180,E1 27919.813,E2 27919.813} C_VEL
LIN {X 0,Y 584.099,Z 49.044,A -85,B 0,C 180,E1 27916.549,E2 27916.549} C_VEL
LIN {X 0,Y 584.099,Z 49.035,A -85,B 0,C 180,E1 27913.26,E2 27913.26} C_VEL
LIN {X 0,Y 584.064,Z 49.038,A -85,B 0,C 180,E1 27910.056,E2 27910.056} C_VEL
LIN {X 0,Y 584.096,Z 49.044,A -85,B 0,C 180,E1 27906.783,E2 27906.783} C_VEL
LIN {X 0,Y 584.091,Z 49.035,A -85,B 0,C 180,E1 27903.533,E2 27903.533} C_VEL
LIN {X 0,Y 584.06,Z 49.039,A -85,B 0,C 180,E1 27900.294,E2 27900.294} C_VEL
LIN {X 0,Y 584.098,Z 49.043,A -85,B 0,C 180,E1 27897.056,E2 27897.056} C_VEL
LIN {X 0,Y 584.08,Z 49.037,A -85,B 0,C 180,E1 27893.809,E2 27893.809} C_VEL
LIN {X 0,Y 584.057,Z 49.04,A -85,B 0,C 180,E1 27890.541,E2 27890.541} C_VEL
LIN {X 0,Y 584.1,Z 49.042,A -85,B 0,C 180,E1 27887.341,E2 27887.341} C_VEL
LIN {X 0,Y 584.058,Z 49.04,A -85,B 0,C 180,E1 27886.709,E2 27886.709} C_VEL
LIN {X 0,Y 583.066,Z 49.163,A -85,B 0,C 180,E1 27885.954,E2 27885.954} C_VEL
LIN {X 0,Y 576.612,Z 49.982,A -85,B 0,C 180,E1 27883.778,E2 27883.778} C_VEL
LIN {X 0,Y 576.154,Z 50.033,A -85,B 0,C 180,E1 27883.281,E2 27883.281} C_VEL
LIN {X 0,Y 576.142,Z 50.027,A -85,B 0,C 180,E1 27880.008,E2 27880.008} C_VEL
LIN {X 0,Y 576.112,Z 50.025,A -85,B 0,C 180,E1 27876.798,E2 27876.798} C_VEL
LIN {X 0,Y 576.159,Z 50.032,A -85,B 0,C 180,E1 27873.564,E2 27873.564} C_VEL
LIN {X 0,Y 576.124,Z 50.026,A -85,B 0,C 180,E1 27870.355,E2 27870.355} C_VEL
LIN {X 0,Y 576.111,Z 50.031,A -85,B 0,C 180,E1 27867.096,E2 27867.096} C_VEL
LIN {X 0,Y 576.16,Z 50.027,A -85,B 0,C 180,E1 27863.964,E2 27863.964} C_VEL
LIN {X 0,Y 576.106,Z 50.03,A -85,B 0,C 180,E1 27860.821,E2 27860.821} C_VEL
LIN {X 0,Y 576.121,Z 50.032,A -85,B 0,C 180,E1 27857.524,E2 27857.524} C_VEL
LIN {X 0,Y 576.148,Z 50.029,A -85,B 0,C 180,E1 27854.357,E2 27854.357} C_VEL
LIN {X 0,Y 576.098,Z 50.032,A -85,B 0,C 180,E1 27851.128,E2 27851.128} C_VEL
LIN {X 0,Y 576.148,Z 50.034,A -85,B 0,C 180,E1 27848.011,E2 27848.011} C_VEL
LIN {X 0,Y 576.108,Z 50.033,A -85,B 0,C 180,E1 27844.939,E2 27844.939} C_VEL
LIN {X 0,Y 576.146,Z 50.292,A -85,B 0,C 180,E1 27842.929,E2 27842.929} C_VEL
LIN {X 0,Y 576.732,Z 54.506,A -85,B 0,C 180,E1 27842.462,E2 27842.462} C_VEL
LIN {X 0,Y 576.904,Z 85.109,A -85,B 0,C 180,E1 27839.334,E2 27839.334} C_VEL
LIN {X 0,Y 576.814,Z 113.031,A -85,B 0,C 180,E1 27836.398,E2 27836.398} C_VEL
LIN {X 0,Y 576.59,Z 139.127,A -85,B 0,C 180,E1 27833.613,E2 27833.613} C_VEL
LIN {X 0,Y 576.321,Z 171.546,A -85,B 0,C 180,E1 27830.184,E2 27830.184} C_VEL
LIN {X 0,Y 576.358,Z 176.148,A -85,B 0,C 180,E1 27829.74,E2 27829.74} C_VEL
LIN {X 0,Y 576.767,Z 183.002,A -85,B 0,C 180,E1 27829.64,E2 27829.64} C_VEL
LIN {X 0,Y 576.569,Z 287.651,A -85,B 0,C 180,E1 27828.307,E2 27828.307} C_VEL
LIN {X 0,Y 576.518,Z 302.469,A -85,B 0,C 180,E1 27827.928,E2 27827.928} C_VEL
LIN {X 0,Y 576.432,Z 315.812,A -85,B 0,C 180,E1 27827.414,E2 27827.414} C_VEL
LIN {X 0,Y 576.297,Z 329.499,A -85,B 0,C 180,E1 27826.691,E2 27826.691} C_VEL
LIN {X 0,Y 576.196,Z 342.111,A -85,B 0,C 180,E1 27825.808,E2 27825.808} C_VEL
LIN {X 0,Y 576.105,Z 353.575,A -85,B 0,C 180,E1 27824.78,E2 27824.78} C_VEL
LIN {X 0,Y 576.029,Z 363.459,A -85,B 0,C 180,E1 27823.653,E2 27823.653} C_VEL
LIN {X 0,Y 575.97,Z 372.49,A -85,B 0,C 180,E1 27822.328,E2 27822.328} C_VEL
LIN {X 0,Y 575.937,Z 379.727,A -85,B 0,C 180,E1 27820.907,E2 27820.907} C_VEL
LIN {X 0,Y 575.922,Z 384.841,A -85,B 0,C 180,E1 27819.492,E2 27819.492} C_VEL
LIN {X 0,Y 575.918,Z 388.151,A -85,B 0,C 180,E1 27818.083,E2 27818.083} C_VEL
LIN {X 0,Y 575.918,Z 389.834,A -85,B 0,C 180,E1 27816.579,E2 27816.579} C_VEL
LIN {X 0,Y 575.916,Z 389.666,A -85,B 0,C 180,E1 27815.079,E2 27815.079} C_VEL
LIN {X 0,Y 575.916,Z 387.897,A -85,B 0,C 180,E1 27813.682,E2 27813.682} C_VEL
LIN {X 0,Y 575.923,Z 384.15,A -85,B 0,C 180,E1 27812.188,E2 27812.188} C_VEL
LIN {X 0,Y 575.94,Z 378.791,A -85,B 0,C 180,E1 27810.795,E2 27810.795} C_VEL
LIN {X 0,Y 575.974,Z 372.008,A -85,B 0,C 180,E1 27809.502,E2 27809.502} C_VEL
LIN {X 0,Y 576.033,Z 363.092,A -85,B 0,C 180,E1 27808.209,E2 27808.209} C_VEL
LIN {X 0,Y 576.117,Z 352.432,A -85,B 0,C 180,E1 27807.015,E2 27807.015} C_VEL
LIN {X 0,Y 576.197,Z 341.059,A -85,B 0,C 180,E1 27806.019,E2 27806.019} C_VEL
LIN {X 0,Y 576.299,Z 328.837,A -85,B 0,C 180,E1 27805.18,E2 27805.18} C_VEL
LIN {X 0,Y 576.435,Z 315.357,A -85,B 0,C 180,E1 27804.475,E2 27804.475} C_VEL
LIN {X 0,Y 576.483,Z 300.745,A -85,B 0,C 180,E1 27803.926,E2 27803.926} C_VEL
LIN {X 0,Y 576.532,Z 285.696,A -85,B 0,C 180,E1 27803.568,E2 27803.568} C_VEL
LIN {X 0,Y 576.539,Z 172.643,A -85,B 0,C 180,E1 27802.131,E2 27802.131} C_VEL
LIN {X 0,Y 576.811,Z 125.065,A -85,B 0,C 180,E1 27799.159,E2 27799.159} C_VEL
LIN {X 0,Y 577.188,Z 76.93,A -85,B 0,C 180,E1 27796.117,E2 27796.117} C_VEL
LIN {X 0,Y 577.168,Z 54.259,A -85,B 0,C 180,E1 27794.686,E2 27794.686} C_VEL
LIN {X 0,Y 576.152,Z 50.306,A -85,B 0,C 180,E1 27794.372,E2 27794.372} C_VEL
LIN {X 0,Y 576.15,Z 50.026,A -85,B 0,C 180,E1 27791.902,E2 27791.902} C_VEL
LIN {X 0,Y 576.226,Z 50.524,A -85,B 0,C 180,E1 27791.65,E2 27791.65} C_VEL
LIN {X 0,Y 577.564,Z 55.905,A -85,B 0,C 180,E1 27791.216,E2 27791.216} C_VEL
LIN {X 0,Y 576.997,Z 107.443,A -85,B 0,C 180,E1 27787.868,E2 27787.868} C_VEL
LIN {X 0,Y 576.605,Z 159.429,A -85,B 0,C 180,E1 27784.59,E2 27784.59} C_VEL
LIN {X 0,Y 576.583,Z 172.508,A -85,B 0,C 180,E1 27783.785,E2 27783.785} C_VEL
LIN {X 0,Y 576.577,Z 287.435,A -85,B 0,C 180,E1 27782.309,E2 27782.309} C_VEL
LIN {X 0,Y 576.526,Z 302.212,A -85,B 0,C 180,E1 27781.938,E2 27781.938} C_VEL
LIN {X 0,Y 576.422,Z 317.445,A -85,B 0,C 180,E1 27781.339,E2 27781.339} C_VEL
LIN {X 0,Y 576.274,Z 331.338,A -85,B 0,C 180,E1 27780.575,E2 27780.575} C_VEL
LIN {X 0,Y 576.199,Z 343.107,A -85,B 0,C 180,E1 27779.728,E2 27779.728} C_VEL
LIN {X 0,Y 576.103,Z 353.985,A -85,B 0,C 180,E1 27778.739,E2 27778.739} C_VEL
LIN {X 0,Y 576.023,Z 364.136,A -85,B 0,C 180,E1 27777.563,E2 27777.563} C_VEL
LIN {X 0,Y 575.972,Z 372.213,A -85,B 0,C 180,E1 27776.374,E2 27776.374} C_VEL
LIN {X 0,Y 575.938,Z 379.649,A -85,B 0,C 180,E1 27774.926,E2 27774.926} C_VEL
LIN {X 0,Y 575.921,Z 384.961,A -85,B 0,C 180,E1 27773.453,E2 27773.453} C_VEL
LIN {X 0,Y 575.918,Z 388.256,A -85,B 0,C 180,E1 27772.018,E2 27772.018} C_VEL
LIN {X 0,Y 575.917,Z 389.855,A -85,B 0,C 180,E1 27770.549,E2 27770.549} C_VEL
LIN {X 0,Y 575.916,Z 389.602,A -85,B 0,C 180,E1 27768.985,E2 27768.985} C_VEL
LIN {X 0,Y 575.919,Z 387.568,A -85,B 0,C 180,E1 27767.519,E2 27767.519} C_VEL
LIN {X 0,Y 575.923,Z 383.599,A -85,B 0,C 180,E1 27766.017,E2 27766.017} C_VEL
LIN {X 0,Y 575.947,Z 377.595,A -85,B 0,C 180,E1 27764.536,E2 27764.536} C_VEL
LIN {X 0,Y 575.984,Z 370.052,A -85,B 0,C 180,E1 27763.19,E2 27763.19} C_VEL
LIN {X 0,Y 576.043,Z 361.588,A -85,B 0,C 180,E1 27762.021,E2 27762.021} C_VEL
LIN {X 0,Y 576.132,Z 350.899,A -85,B 0,C 180,E1 27760.865,E2 27760.865} C_VEL
LIN {X 0,Y 576.225,Z 338.877,A -85,B 0,C 180,E1 27759.854,E2 27759.854} C_VEL
LIN {X 0,Y 576.34,Z 326.29,A -85,B 0,C 180,E1 27759.032,E2 27759.032} C_VEL
LIN {X 0,Y 576.461,Z 312.271,A -85,B 0,C 180,E1 27758.341,E2 27758.341} C_VEL
LIN {X 0,Y 576.553,Z 296.855,A -85,B 0,C 180,E1 27757.814,E2 27757.814} C_VEL
LIN {X 0,Y 576.61,Z 281.374,A -85,B 0,C 180,E1 27757.502,E2 27757.502} C_VEL
LIN {X 0,Y 576.537,Z 177.338,A -85,B 0,C 180,E1 27756.194,E2 27756.194} C_VEL
LIN {X 0,Y 576.352,Z 175.693,A -85,B 0,C 180,E1 27756.146,E2 27756.146} C_VEL
LIN {X 0,Y 576.544,Z 145.038,A -85,B 0,C 180,E1 27752.927,E2 27752.927} C_VEL
LIN {X 0,Y 576.953,Z 115.044,A -85,B 0,C 180,E1 27749.655,E2 27749.655} C_VEL
LIN {X 0,Y 577.363,Z 84.886,A -85,B 0,C 180,E1 27746.317,E2 27746.317} C_VEL
LIN {X 0,Y 577.78,Z 57.676,A -85,B 0,C 180,E1 27743.234,E2 27743.234} C_VEL
LIN {X 0,Y 577.036,Z 53.644,A -85,B 0,C 180,E1 27742.731,E2 27742.731} C_VEL
LIN {X 0,Y 576.164,Z 50.127,A -85,B 0,C 180,E1 27742.229,E2 27742.229} C_VEL
LIN {X 0,Y 576.112,Z 50.033,A -85,B 0,C 180,E1 27739.043,E2 27739.043} C_VEL
LIN {X 0,Y 576.156,Z 50.033,A -85,B 0,C 180,E1 27735.811,E2 27735.811} C_VEL
LIN {X 0,Y 576.126,Z 50.029,A -85,B 0,C 180,E1 27732.631,E2 27732.631} C_VEL
LIN {X 0,Y 576.109,Z 50.03,A -85,B 0,C 180,E1 27729.389,E2 27729.389} C_VEL
LIN {X 0,Y 576.162,Z 50.032,A -85,B 0,C 180,E1 27726.177,E2 27726.177} C_VEL
LIN {X 0,Y 576.11,Z 50.03,A -85,B 0,C 180,E1 27722.985,E2 27722.985} C_VEL
LIN {X 0,Y 576.11,Z 50.032,A -85,B 0,C 180,E1 27719.702,E2 27719.702} C_VEL
LIN {X 0,Y 576.16,Z 50.03,A -85,B 0,C 180,E1 27716.518,E2 27716.518} C_VEL
LIN {X 0,Y 576.099,Z 50.031,A -85,B 0,C 180,E1 27713.323,E2 27713.323} C_VEL
LIN {X 0,Y 576.121,Z 50.033,A -85,B 0,C 180,E1 27710.107,E2 27710.107} C_VEL
LIN {X 0,Y 576.118,Z 50.031,A -85,B 0,C 180,E1 27707.063,E2 27707.063} C_VEL
LIN {X 0,Y 576.095,Z 50.032,A -85,B 0,C 180,E1 27703.878,E2 27703.878} C_VEL
LIN {X 0,Y 576.159,Z 50.031,A -85,B 0,C 180,E1 27700.743,E2 27700.743} C_VEL
LIN {X 0,Y 576.089,Z 50.032,A -85,B 0,C 180,E1 27697.661,E2 27697.661} C_VEL
LIN {X 0,Y 576.109,Z 50.033,A -85,B 0,C 180,E1 27694.396,E2 27694.396} C_VEL
LIN {X 0,Y 576.111,Z 50.032,A -85,B 0,C 180,E1 27691.38,E2 27691.38} C_VEL
LIN {X 0,Y 576.084,Z 50.033,A -85,B 0,C 180,E1 27688.155,E2 27688.155} C_VEL
LIN {X 0,Y 576.152,Z 50.034,A -85,B 0,C 180,E1 27684.996,E2 27684.996} C_VEL
LIN {X 0,Y 576.086,Z 50.033,A -85,B 0,C 180,E1 27681.835,E2 27681.835} C_VEL
LIN {X 0,Y 576.083,Z 50.034,A -85,B 0,C 180,E1 27678.471,E2 27678.471} C_VEL
LIN {X 0,Y 576.145,Z 50.033,A -85,B 0,C 180,E1 27675.344,E2 27675.344} C_VEL
LIN {X 0,Y 576.083,Z 50.034,A -85,B 0,C 180,E1 27672.174,E2 27672.174} C_VEL
LIN {X 0,Y 576.111,Z 50.034,A -85,B 0,C 180,E1 27668.966,E2 27668.966} C_VEL
LIN {X 0,Y 576.108,Z 50.035,A -85,B 0,C 180,E1 27665.917,E2 27665.917} C_VEL
LIN {X 0,Y 576.088,Z 50.032,A -85,B 0,C 180,E1 27662.668,E2 27662.668} C_VEL
LIN {X 0,Y 576.163,Z 50.315,A -85,B 0,C 180,E1 27661.181,E2 27661.181} C_VEL
LIN {X 0,Y 578.549,Z 58.5,A -85,B 0,C 180,E1 27660.415,E2 27660.415} C_VEL
LIN {X 0,Y 578.193,Z 97.595,A -85,B 0,C 180,E1 27657.666,E2 27657.666} C_VEL
LIN {X 0,Y 577.86,Z 145.038,A -85,B 0,C 180,E1 27654.428,E2 27654.428} C_VEL
LIN {X 0,Y 577.807,Z 158.185,A -85,B 0,C 180,E1 27653.558,E2 27653.558} C_VEL
LIN {X 0,Y 578.375,Z 164.383,A -85,B 0,C 180,E1 27653.448,E2 27653.448} C_VEL
LIN {X 0,Y 577.843,Z 367.301,A -85,B 0,C 180,E1 27650.777,E2 27650.777} C_VEL
LIN {X 0,Y 577.689,Z 386.295,A -85,B 0,C 180,E1 27650.337,E2 27650.337} C_VEL
LIN {X 0,Y 577.497,Z 404.387,A -85,B 0,C 180,E1 27649.732,E2 27649.732} C_VEL
LIN {X 0,Y 577.268,Z 422.333,A -85,B 0,C 180,E1 27648.936,E2 27648.936} C_VEL
LIN {X 0,Y 577.028,Z 439.577,A -85,B 0,C 180,E1 27647.965,E2 27647.965} C_VEL
LIN {X 0,Y 576.797,Z 455.181,A -85,B 0,C 180,E1 27646.888,E2 27646.888} C_VEL
LIN {X 0,Y 576.571,Z 470.107,A -85,B 0,C 180,E1 27645.645,E2 27645.645} C_VEL
LIN {X 0,Y 576.37,Z 483.94,A -85,B 0,C 180,E1 27644.261,E2 27644.261} C_VEL
LIN {X 0,Y 576.207,Z 496.683,A -85,B 0,C 180,E1 27642.732,E2 27642.732} C_VEL
LIN {X 0,Y 576.086,Z 507.863,A -85,B 0,C 180,E1 27641.108,E2 27641.108} C_VEL
LIN {X 0,Y 575.999,Z 517.506,A -85,B 0,C 180,E1 27639.392,E2 27639.392} C_VEL
LIN {X 0,Y 575.955,Z 525.176,A -85,B 0,C 180,E1 27637.682,E2 27637.682} C_VEL
LIN {X 0,Y 575.928,Z 531.471,A -85,B 0,C 180,E1 27635.86,E2 27635.86} C_VEL
LIN {X 0,Y 575.914,Z 535.874,A -85,B 0,C 180,E1 27634.083,E2 27634.083} C_VEL
LIN {X 0,Y 575.913,Z 538.79,A -85,B 0,C 180,E1 27632.19,E2 27632.19} C_VEL
LIN {X 0,Y 575.907,Z 539.939,A -85,B 0,C 180,E1 27630.299,E2 27630.299} C_VEL
LIN {X 0,Y 575.913,Z 539.349,A -85,B 0,C 180,E1 27628.409,E2 27628.409} C_VEL
LIN {X 0,Y 575.908,Z 537.006,A -85,B 0,C 180,E1 27626.517,E2 27626.517} C_VEL
LIN {X 0,Y 575.923,Z 533.099,A -85,B 0,C 180,E1 27624.721,E2 27624.721} C_VEL
LIN {X 0,Y 575.941,Z 527.47,A -85,B 0,C 180,E1 27622.921,E2 27622.921} C_VEL
LIN {X 0,Y 575.982,Z 520.43,A -85,B 0,C 180,E1 27621.214,E2 27621.214} C_VEL
LIN {X 0,Y 576.054,Z 511.52,A -85,B 0,C 180,E1 27619.5,E2 27619.5} C_VEL
LIN {X 0,Y 576.157,Z 501.156,A -85,B 0,C 180,E1 27617.88,E2 27617.88} C_VEL
LIN {X 0,Y 576.307,Z 488.951,A -85,B 0,C 180,E1 27616.304,E2 27616.304} C_VEL
LIN {X 0,Y 576.498,Z 475.587,A -85,B 0,C 180,E1 27614.87,E2 27614.87} C_VEL
LIN {X 0,Y 576.719,Z 460.615,A -85,B 0,C 180,E1 27613.534,E2 27613.534} C_VEL
LIN {X 0,Y 576.96,Z 444.448,A -85,B 0,C 180,E1 27612.347,E2 27612.347} C_VEL
LIN {X 0,Y 577.199,Z 428.03,A -85,B 0,C 180,E1 27611.36,E2 27611.36} C_VEL
LIN {X 0,Y 577.428,Z 410.837,A -85,B 0,C 180,E1 27610.53,E2 27610.53} C_VEL
LIN {X 0,Y 577.636,Z 392.669,A -85,B 0,C 180,E1 27609.856,E2 27609.856} C_VEL
LIN {X 0,Y 577.797,Z 374.196,A -85,B 0,C 180,E1 27609.362,E2 27609.362} C_VEL
LIN {X 0,Y 577.898,Z 354.214,A -85,B 0,C 180,E1 27609.028,E2 27609.028} C_VEL
LIN {X 0,Y 578.25,Z 156.572,A -85,B 0,C 180,E1 27606.443,E2 27606.443} C_VEL
LIN {X 0,Y 578.166,Z 149.236,A -85,B 0,C 180,E1 27606.182,E2 27606.182} C_VEL
LIN {X 0,Y 578.599,Z 80.934,A -85,B 0,C 180,E1 27603.413,E2 27603.413} C_VEL
LIN {X 0,Y 578.592,Z 57.057,A -85,B 0,C 180,E1 27602.438,E2 27602.438} C_VEL
LIN {X 0,Y 576.215,Z 50.484,A -85,B 0,C 180,E1 27602.013,E2 27602.013} C_VEL
LIN {X 0,Y 576.146,Z 50.029,A -85,B 0,C 180,E1 27601.835,E2 27601.835} C_VEL
LIN {X 0,Y 576.158,Z 50.025,A -85,B 0,C 180,E1 27598.511,E2 27598.511} C_VEL
LIN {X 0,Y 576.141,Z 50.029,A -85,B 0,C 180,E1 27595.171,E2 27595.171} C_VEL
LIN {X 0,Y 576.156,Z 50.033,A -85,B 0,C 180,E1 27591.846,E2 27591.846} C_VEL
LIN {X 0,Y 576.153,Z 50.026,A -85,B 0,C 180,E1 27588.479,E2 27588.479} C_VEL
LIN {X 0,Y 576.139,Z 50.027,A -85,B 0,C 180,E1 27585.205,E2 27585.205} C_VEL
LIN {X 0,Y 576.158,Z 50.032,A -85,B 0,C 180,E1 27581.888,E2 27581.888} C_VEL
LIN {X 0,Y 576.152,Z 50.027,A -85,B 0,C 180,E1 27578.536,E2 27578.536} C_VEL
LIN {X 0,Y 576.138,Z 50.025,A -85,B 0,C 180,E1 27575.303,E2 27575.303} C_VEL
LIN {X 0,Y 576.145,Z 50.03,A -85,B 0,C 180,E1 27571.941,E2 27571.941} C_VEL
LIN {X 0,Y 576.153,Z 50.027,A -85,B 0,C 180,E1 27568.731,E2 27568.731} C_VEL
LIN {X 0,Y 576.135,Z 50.026,A -85,B 0,C 180,E1 27565.492,E2 27565.492} C_VEL
LIN {X 0,Y 576.141,Z 50.031,A -85,B 0,C 180,E1 27562.123,E2 27562.123} C_VEL
LIN {X 0,Y 576.155,Z 50.027,A -85,B 0,C 180,E1 27558.831,E2 27558.831} C_VEL
LIN {X 0,Y 576.135,Z 50.026,A -85,B 0,C 180,E1 27555.603,E2 27555.603} C_VEL
LIN {X 0,Y 576.131,Z 50.03,A -85,B 0,C 180,E1 27552.223,E2 27552.223} C_VEL
LIN {X 0,Y 576.157,Z 50.027,A -85,B 0,C 180,E1 27548.985,E2 27548.985} C_VEL
LIN {X 0,Y 576.132,Z 50.026,A -85,B 0,C 180,E1 27545.777,E2 27545.777} C_VEL
LIN {X 0,Y 576.131,Z 50.031,A -85,B 0,C 180,E1 27542.486,E2 27542.486} C_VEL
LIN {X 0,Y 576.159,Z 50.025,A -85,B 0,C 180,E1 27539.304,E2 27539.304} C_VEL
LIN {X 0,Y 576.122,Z 50.027,A -85,B 0,C 180,E1 27536.119,E2 27536.119} C_VEL
LIN {X 0,Y 576.137,Z 50.031,A -85,B 0,C 180,E1 27532.822,E2 27532.822} C_VEL
LIN {X 0,Y 576.158,Z 50.025,A -85,B 0,C 180,E1 27529.602,E2 27529.602} C_VEL
LIN {X 0,Y 576.117,Z 50.027,A -85,B 0,C 180,E1 27526.347,E2 27526.347} C_VEL
LIN {X 0,Y 576.154,Z 50.033,A -85,B 0,C 180,E1 27523.281,E2 27523.281} C_VEL
LIN {X 0,Y 575.129,Z 50.154,A -85,B 0,C 180,E1 27522.515,E2 27522.515} C_VEL
LIN {X 0,Y 568.727,Z 50.95,A -85,B 0,C 180,E1 27520.365,E2 27520.365} C_VEL
LIN {X 0,Y 568.218,Z 51.016,A -85,B 0,C 180,E1 27519.806,E2 27519.806} C_VEL
LIN {X 0,Y 568.173,Z 51.012,A -85,B 0,C 180,E1 27516.565,E2 27516.565} C_VEL
LIN {X 0,Y 568.191,Z 51.021,A -85,B 0,C 180,E1 27513.225,E2 27513.225} C_VEL
LIN {X 0,Y 568.223,Z 51.013,A -85,B 0,C 180,E1 27509.963,E2 27509.963} C_VEL
LIN {X 0,Y 568.17,Z 51.019,A -85,B 0,C 180,E1 27506.707,E2 27506.707} C_VEL
LIN {X 0,Y 568.181,Z 51.021,A -85,B 0,C 180,E1 27503.362,E2 27503.362} C_VEL
LIN {X 0,Y 568.22,Z 51.017,A -85,B 0,C 180,E1 27500.17,E2 27500.17} C_VEL
LIN {X 0,Y 568.166,Z 51.019,A -85,B 0,C 180,E1 27496.911,E2 27496.911} C_VEL
LIN {X 0,Y 568.182,Z 51.02,A -85,B 0,C 180,E1 27493.614,E2 27493.614} C_VEL
LIN {X 0,Y 568.217,Z 51.019,A -85,B 0,C 180,E1 27490.355,E2 27490.355} C_VEL
LIN {X 0,Y 568.16,Z 51.022,A -85,B 0,C 180,E1 27487.128,E2 27487.128} C_VEL
LIN {X 0,Y 568.179,Z 51.026,A -85,B 0,C 180,E1 27483.838,E2 27483.838} C_VEL
LIN {X 0,Y 568.204,Z 51.313,A -85,B 0,C 180,E1 27483.111,E2 27483.111} C_VEL
LIN {X 0,Y 568.977,Z 56.025,A -85,B 0,C 180,E1 27482.588,E2 27482.588} C_VEL
LIN {X 0,Y 569.113,Z 84.867,A -85,B 0,C 180,E1 27479.633,E2 27479.633} C_VEL
LIN {X 0,Y 569.061,Z 114.044,A -85,B 0,C 180,E1 27476.577,E2 27476.577} C_VEL
LIN {X 0,Y 568.829,Z 138.723,A -85,B 0,C 180,E1 27473.931,E2 27473.931} C_VEL
LIN {X 0,Y 568.567,Z 165.15,A -85,B 0,C 180,E1 27471.076,E2 27471.076} C_VEL
LIN {X 0,Y 568.469,Z 176.113,A -85,B 0,C 180,E1 27469.937,E2 27469.937} C_VEL
LIN {X 0,Y 568.994,Z 182.943,A -85,B 0,C 180,E1 27469.831,E2 27469.831} C_VEL
LIN {X 0,Y 568.751,Z 287.617,A -85,B 0,C 180,E1 27468.48,E2 27468.48} C_VEL
LIN {X 0,Y 568.683,Z 302.191,A -85,B 0,C 180,E1 27468.104,E2 27468.104} C_VEL
LIN {X 0,Y 568.566,Z 316.298,A -85,B 0,C 180,E1 27467.552,E2 27467.552} C_VEL
LIN {X 0,Y 568.403,Z 329.865,A -85,B 0,C 180,E1 27466.819,E2 27466.819} C_VEL
LIN {X 0,Y 568.268,Z 342.983,A -85,B 0,C 180,E1 27465.877,E2 27465.877} C_VEL
LIN {X 0,Y 568.151,Z 354.296,A -85,B 0,C 180,E1 27464.829,E2 27464.829} C_VEL
LIN {X 0,Y 568.055,Z 364.034,A -85,B 0,C 180,E1 27463.686,E2 27463.686} C_VEL
LIN {X 0,Y 567.985,Z 372.591,A -85,B 0,C 180,E1 27462.401,E2 27462.401} C_VEL
LIN {X 0,Y 567.943,Z 379.801,A -85,B 0,C 180,E1 27460.96,E2 27460.96} C_VEL
LIN {X 0,Y 567.923,Z 384.891,A -85,B 0,C 180,E1 27459.525,E2 27459.525} C_VEL
LIN {X 0,Y 567.919,Z 388.177,A -85,B 0,C 180,E1 27458.096,E2 27458.096} C_VEL
LIN {X 0,Y 567.918,Z 389.845,A -85,B 0,C 180,E1 27456.57,E2 27456.57} C_VEL
LIN {X 0,Y 567.916,Z 389.655,A -85,B 0,C 180,E1 27455.049,E2 27455.049} C_VEL
LIN {X 0,Y 567.916,Z 387.863,A -85,B 0,C 180,E1 27453.633,E2 27453.633} C_VEL
LIN {X 0,Y 567.926,Z 384.1,A -85,B 0,C 180,E1 27452.118,E2 27452.118} C_VEL
LIN {X 0,Y 567.947,Z 378.714,A -85,B 0,C 180,E1 27450.705,E2 27450.705} C_VEL
LIN {X 0,Y 567.991,Z 371.903,A -85,B 0,C 180,E1 27449.394,E2 27449.394} C_VEL
LIN {X 0,Y 568.067,Z 362.968,A -85,B 0,C 180,E1 27448.083,E2 27448.083} C_VEL
LIN {X 0,Y 568.176,Z 352.271,A -85,B 0,C 180,E1 27446.872,E2 27446.872} C_VEL
LIN {X 0,Y 568.283,Z 340.208,A -85,B 0,C 180,E1 27445.812,E2 27445.812} C_VEL
LIN {X 0,Y 568.427,Z 327.571,A -85,B 0,C 180,E1 27444.954,E2 27444.954} C_VEL
LIN {X 0,Y 568.584,Z 313.829,A -85,B 0,C 180,E1 27444.247,E2 27444.247} C_VEL
LIN {X 0,Y 568.654,Z 299.046,A -85,B 0,C 180,E1 27443.706,E2 27443.706} C_VEL
LIN {X 0,Y 568.732,Z 283.304,A -85,B 0,C 180,E1 27443.353,E2 27443.353} C_VEL
LIN {X 0,Y 568.77,Z 173.361,A -85,B 0,C 180,E1 27441.951,E2 27441.951} C_VEL
LIN {X 0,Y 568.692,Z 169.639,A -85,B 0,C 180,E1 27441.761,E2 27441.761} C_VEL
LIN {X 0,Y 569.187,Z 119.343,A -85,B 0,C 180,E1 27438.55,E2 27438.55} C_VEL
LIN {X 0,Y 569.504,Z 72.092,A -85,B 0,C 180,E1 27435.563,E2 27435.563} C_VEL
LIN {X 0,Y 569.47,Z 56.238,A -85,B 0,C 180,E1 27434.563,E2 27434.563} C_VEL
LIN {X 0,Y 568.251,Z 51.477,A -85,B 0,C 180,E1 27434.199,E2 27434.199} C_VEL
LIN {X 0,Y 568.198,Z 51.025,A -85,B 0,C 180,E1 27433.962,E2 27433.962} C_VEL
LIN {X 0,Y 568.25,Z 51.267,A -85,B 0,C 180,E1 27431.986,E2 27431.986} C_VEL
LIN {X 0,Y 569.737,Z 56.342,A -85,B 0,C 180,E1 27431.532,E2 27431.532} C_VEL
LIN {X 0,Y 570.025,Z 59.661,A -85,B 0,C 180,E1 27431.298,E2 27431.298} C_VEL
LIN {X 0,Y 569.359,Z 110.219,A -85,B 0,C 180,E1 27427.98,E2 27427.98} C_VEL
LIN {X 0,Y 568.786,Z 161.621,A -85,B 0,C 180,E1 27424.656,E2 27424.656} C_VEL
LIN {X 0,Y 568.758,Z 172.391,A -85,B 0,C 180,E1 27423.984,E2 27423.984} C_VEL
LIN {X 0,Y 568.983,Z 186.71,A -85,B 0,C 180,E1 27423.783,E2 27423.783} C_VEL
LIN {X 0,Y 568.759,Z 287.475,A -85,B 0,C 180,E1 27422.481,E2 27422.481} C_VEL
LIN {X 0,Y 568.696,Z 301.874,A -85,B 0,C 180,E1 27422.116,E2 27422.116} C_VEL
LIN {X 0,Y 568.563,Z 316.598,A -85,B 0,C 180,E1 27421.538,E2 27421.538} C_VEL
LIN {X 0,Y 568.406,Z 329.502,A -85,B 0,C 180,E1 27420.839,E2 27420.839} C_VEL
LIN {X 0,Y 568.287,Z 342.02,A -85,B 0,C 180,E1 27419.956,E2 27419.956} C_VEL
LIN {X 0,Y 568.154,Z 354.193,A -85,B 0,C 180,E1 27418.842,E2 27418.842} C_VEL
LIN {X 0,Y 568.052,Z 364.294,A -85,B 0,C 180,E1 27417.65,E2 27417.65} C_VEL
LIN {X 0,Y 567.983,Z 372.732,A -85,B 0,C 180,E1 27416.373,E2 27416.373} C_VEL
LIN {X 0,Y 567.943,Z 379.85,A -85,B 0,C 180,E1 27414.948,E2 27414.948} C_VEL
LIN {X 0,Y 567.923,Z 385.265,A -85,B 0,C 180,E1 27413.4,E2 27413.4} C_VEL
LIN {X 0,Y 567.916,Z 388.481,A -85,B 0,C 180,E1 27411.904,E2 27411.904} C_VEL
LIN {X 0,Y 567.916,Z 389.906,A -85,B 0,C 180,E1 27410.407,E2 27410.407} C_VEL
LIN {X 0,Y 567.916,Z 389.492,A -85,B 0,C 180,E1 27408.818,E2 27408.818} C_VEL
LIN {X 0,Y 567.919,Z 387.06,A -85,B 0,C 180,E1 27407.236,E2 27407.236} C_VEL
LIN {X 0,Y 567.93,Z 382.931,A -85,B 0,C 180,E1 27405.77,E2 27405.77} C_VEL
LIN {X 0,Y 567.958,Z 377.012,A -85,B 0,C 180,E1 27404.339,E2 27404.339} C_VEL
LIN {X 0,Y 568.015,Z 368.97,A -85,B 0,C 180,E1 27402.923,E2 27402.923} C_VEL
LIN {X 0,Y 568.101,Z 359.268,A -85,B 0,C 180,E1 27401.63,E2 27401.63} C_VEL
LIN {X 0,Y 568.213,Z 348.578,A -85,B 0,C 180,E1 27400.521,E2 27400.521} C_VEL
LIN {X 0,Y 568.338,Z 336.808,A -85,B 0,C 180,E1 27399.558,E2 27399.558} C_VEL
LIN {X 0,Y 568.5,Z 323.144,A -85,B 0,C 180,E1 27398.7,E2 27398.7} C_VEL
LIN {X 0,Y 568.639,Z 308.446,A -85,B 0,C 180,E1 27398.026,E2 27398.026} C_VEL
LIN {X 0,Y 568.736,Z 293.939,A -85,B 0,C 180,E1 27397.571,E2 27397.571} C_VEL
LIN {X 0,Y 568.807,Z 278.702,A -85,B 0,C 180,E1 27397.291,E2 27397.291} C_VEL
LIN {X 0,Y 568.775,Z 178.216,A -85,B 0,C 180,E1 27396.013,E2 27396.013} C_VEL
LIN {X 0,Y 568.472,Z 175.646,A -85,B 0,C 180,E1 27395.946,E2 27395.946} C_VEL
LIN {X 0,Y 568.784,Z 146.799,A -85,B 0,C 180,E1 27392.831,E2 27392.831} C_VEL
LIN {X 0,Y 569.291,Z 116.332,A -85,B 0,C 180,E1 27389.457,E2 27389.457} C_VEL
LIN {X 0,Y 569.763,Z 86.601,A -85,B 0,C 180,E1 27386.134,E2 27386.134} C_VEL
LIN {X 0,Y 570.257,Z 59.872,A -85,B 0,C 180,E1 27383.071,E2 27383.071} C_VEL
LIN {X 0,Y 568.241,Z 51.152,A -85,B 0,C 180,E1 27381.903,E2 27381.903} C_VEL
LIN {X 0,Y 568.18,Z 51.021,A -85,B 0,C 180,E1 27378.68,E2 27378.68} C_VEL
LIN {X 0,Y 568.177,Z 51.021,A -85,B 0,C 180,E1 27375.306,E2 27375.306} C_VEL
LIN {X 0,Y 568.222,Z 51.02,A -85,B 0,C 180,E1 27372.087,E2 27372.087} C_VEL
LIN {X 0,Y 568.171,Z 51.018,A -85,B 0,C 180,E1 27368.909,E2 27368.909} C_VEL
LIN {X 0,Y 568.172,Z 51.022,A -85,B 0,C 180,E1 27365.554,E2 27365.554} C_VEL
LIN {X 0,Y 568.222,Z 51.02,A -85,B 0,C 180,E1 27362.32,E2 27362.32} C_VEL
LIN {X 0,Y 568.164,Z 51.02,A -85,B 0,C 180,E1 27359.194,E2 27359.194} C_VEL
LIN {X 0,Y 568.175,Z 51.022,A -85,B 0,C 180,E1 27355.863,E2 27355.863} C_VEL
LIN {X 0,Y 568.21,Z 51.019,A -85,B 0,C 180,E1 27352.721,E2 27352.721} C_VEL
LIN {X 0,Y 568.157,Z 51.021,A -85,B 0,C 180,E1 27349.557,E2 27349.557} C_VEL
LIN {X 0,Y 568.199,Z 51.022,A -85,B 0,C 180,E1 27346.361,E2 27346.361} C_VEL
LIN {X 0,Y 568.172,Z 51.019,A -85,B 0,C 180,E1 27343.226,E2 27343.226} C_VEL
LIN {X 0,Y 568.155,Z 51.021,A -85,B 0,C 180,E1 27339.93,E2 27339.93} C_VEL
LIN {X 0,Y 568.22,Z 51.021,A -85,B 0,C 180,E1 27336.787,E2 27336.787} C_VEL
LIN {X 0,Y 568.154,Z 51.021,A -85,B 0,C 180,E1 27333.605,E2 27333.605} C_VEL
LIN {X 0,Y 568.153,Z 51.022,A -85,B 0,C 180,E1 27330.246,E2 27330.246} C_VEL
LIN {X 0,Y 568.202,Z 51.022,A -85,B 0,C 180,E1 27327.181,E2 27327.181} C_VEL
LIN {X 0,Y 568.143,Z 51.022,A -85,B 0,C 180,E1 27323.999,E2 27323.999} C_VEL
LIN {X 0,Y 568.17,Z 51.023,A -85,B 0,C 180,E1 27320.742,E2 27320.742} C_VEL
LIN {X 0,Y 568.153,Z 51.024,A -85,B 0,C 180,E1 27317.758,E2 27317.758} C_VEL
LIN {X 0,Y 568.144,Z 51.023,A -85,B 0,C 180,E1 27314.461,E2 27314.461} C_VEL
LIN {X 0,Y 568.217,Z 51.02,A -85,B 0,C 180,E1 27311.29,E2 27311.29} C_VEL
LIN {X 0,Y 568.151,Z 51.024,A -85,B 0,C 180,E1 27308.126,E2 27308.126} C_VEL
LIN {X 0,Y 568.153,Z 51.024,A -85,B 0,C 180,E1 27304.73,E2 27304.73} C_VEL
LIN {X 0,Y 568.244,Z 51.22,A -85,B 0,C 180,E1 27301.58,E2 27301.58} C_VEL
LIN {X 0,Y 570.348,Z 57.931,A -85,B 0,C 180,E1 27300.907,E2 27300.907} C_VEL
LIN {X 0,Y 571.211,Z 61.098,A -85,B 0,C 180,E1 27300.622,E2 27300.622} C_VEL
LIN {X 0,Y 570.73,Z 96.066,A -85,B 0,C 180,E1 27298.116,E2 27298.116} C_VEL
LIN {X 0,Y 570.323,Z 142.942,A -85,B 0,C 180,E1 27294.883,E2 27294.883} C_VEL
LIN {X 0,Y 570.268,Z 158.21,A -85,B 0,C 180,E1 27293.874,E2 27293.874} C_VEL
LIN {X 0,Y 571.017,Z 165.074,A -85,B 0,C 180,E1 27293.755,E2 27293.755} C_VEL
LIN {X 0,Y 570.361,Z 367.301,A -85,B 0,C 180,E1 27291.062,E2 27291.062} C_VEL
LIN {X 0,Y 570.168,Z 386.337,A -85,B 0,C 180,E1 27290.616,E2 27290.616} C_VEL
LIN {X 0,Y 569.928,Z 404.384,A -85,B 0,C 180,E1 27290.005,E2 27290.005} C_VEL
LIN {X 0,Y 569.643,Z 422.113,A -85,B 0,C 180,E1 27289.21,E2 27289.21} C_VEL
LIN {X 0,Y 569.351,Z 438.76,A -85,B 0,C 180,E1 27288.269,E2 27288.269} C_VEL
LIN {X 0,Y 569.053,Z 454.619,A -85,B 0,C 180,E1 27287.169,E2 27287.169} C_VEL
LIN {X 0,Y 568.768,Z 469.55,A -85,B 0,C 180,E1 27285.917,E2 27285.917} C_VEL
LIN {X 0,Y 568.522,Z 483.014,A -85,B 0,C 180,E1 27284.566,E2 27284.566} C_VEL
LIN {X 0,Y 568.31,Z 495.911,A -85,B 0,C 180,E1 27283.015,E2 27283.015} C_VEL
LIN {X 0,Y 568.143,Z 507.227,A -85,B 0,C 180,E1 27281.368,E2 27281.368} C_VEL
LIN {X 0,Y 568.032,Z 516.991,A -85,B 0,C 180,E1 27279.627,E2 27279.627} C_VEL
LIN {X 0,Y 567.967,Z 524.771,A -85,B 0,C 180,E1 27277.893,E2 27277.893} C_VEL
LIN {X 0,Y 567.934,Z 531.11,A -85,B 0,C 180,E1 27276.064,E2 27276.064} C_VEL
LIN {X 0,Y 567.913,Z 535.875,A -85,B 0,C 180,E1 27274.14,E2 27274.14} C_VEL
LIN {X 0,Y 567.913,Z 538.791,A -85,B 0,C 180,E1 27272.221,E2 27272.221} C_VEL
LIN {X 0,Y 567.907,Z 539.939,A -85,B 0,C 180,E1 27270.303,E2 27270.303} C_VEL
LIN {X 0,Y 567.914,Z 539.416,A -85,B 0,C 180,E1 27268.488,E2 27268.488} C_VEL
LIN {X 0,Y 567.909,Z 537.165,A -85,B 0,C 180,E1 27266.569,E2 27266.569} C_VEL
LIN {X 0,Y 567.925,Z 533.353,A -85,B 0,C 180,E1 27264.748,E2 27264.748} C_VEL
LIN {X 0,Y 567.948,Z 527.822,A -85,B 0,C 180,E1 27262.922,E2 27262.922} C_VEL
LIN {X 0,Y 568.005,Z 520.43,A -85,B 0,C 180,E1 27261.09,E2 27261.09} C_VEL
LIN {X 0,Y 568.094,Z 511.521,A -85,B 0,C 180,E1 27259.351,E2 27259.351} C_VEL
LIN {X 0,Y 568.231,Z 501.158,A -85,B 0,C 180,E1 27257.708,E2 27257.708} C_VEL
LIN {X 0,Y 568.413,Z 489.359,A -85,B 0,C 180,E1 27256.16,E2 27256.16} C_VEL
LIN {X 0,Y 568.649,Z 476.092,A -85,B 0,C 180,E1 27254.709,E2 27254.709} C_VEL
LIN {X 0,Y 568.926,Z 461.234,A -85,B 0,C 180,E1 27253.355,E2 27253.355} C_VEL
LIN {X 0,Y 569.234,Z 445.327,A -85,B 0,C 180,E1 27252.157,E2 27252.157} C_VEL
LIN {X 0,Y 569.543,Z 428.176,A -85,B 0,C 180,E1 27251.108,E2 27251.108} C_VEL
LIN {X 0,Y 569.834,Z 410.841,A -85,B 0,C 180,E1 27250.26,E2 27250.26} C_VEL
LIN {X 0,Y 570.097,Z 392.565,A -85,B 0,C 180,E1 27249.574,E2 27249.574} C_VEL
LIN {X 0,Y 570.302,Z 374.031,A -85,B 0,C 180,E1 27249.075,E2 27249.075} C_VEL
LIN {X 0,Y 570.428,Z 353.959,A -85,B 0,C 180,E1 27248.737,E2 27248.737} C_VEL
LIN {X 0,Y 570.891,Z 157.431,A -85,B 0,C 180,E1 27246.141,E2 27246.141} C_VEL
LIN {X 0,Y 570.696,Z 152.962,A -85,B 0,C 180,E1 27246.018,E2 27246.018} C_VEL
LIN {X 0,Y 571.204,Z 74.786,A -85,B 0,C 180,E1 27242.845,E2 27242.845} C_VEL
LIN {X 0,Y 571.298,Z 59.67,A -85,B 0,C 180,E1 27242.215,E2 27242.215} C_VEL
LIN {X 0,Y 568.31,Z 51.616,A -85,B 0,C 180,E1 27241.698,E2 27241.698} C_VEL
LIN {X 0,Y 568.217,Z 51.022,A -85,B 0,C 180,E1 27241.521,E2 27241.521} C_VEL
LIN {X 0,Y 568.209,Z 51.017,A -85,B 0,C 180,E1 27238.203,E2 27238.203} C_VEL
LIN {X 0,Y 568.206,Z 51.015,A -85,B 0,C 180,E1 27234.91,E2 27234.91} C_VEL
LIN {X 0,Y 568.211,Z 51.021,A -85,B 0,C 180,E1 27231.541,E2 27231.541} C_VEL
LIN {X 0,Y 568.21,Z 51.018,A -85,B 0,C 180,E1 27228.253,E2 27228.253} C_VEL
LIN {X 0,Y 568.21,Z 51.014,A -85,B 0,C 180,E1 27224.98,E2 27224.98} C_VEL
LIN {X 0,Y 568.202,Z 51.018,A -85,B 0,C 180,E1 27221.596,E2 27221.596} C_VEL
LIN {X 0,Y 568.215,Z 51.019,A -85,B 0,C 180,E1 27218.272,E2 27218.272} C_VEL
LIN {X 0,Y 568.22,Z 51.012,A -85,B 0,C 180,E1 27214.881,E2 27214.881} C_VEL
LIN {X 0,Y 568.195,Z 51.016,A -85,B 0,C 180,E1 27211.606,E2 27211.606} C_VEL
LIN {X 0,Y 568.221,Z 51.02,A -85,B 0,C 180,E1 27208.366,E2 27208.366} C_VEL
LIN {X 0,Y 568.217,Z 51.014,A -85,B 0,C 180,E1 27204.981,E2 27204.981} C_VEL
LIN {X 0,Y 568.192,Z 51.017,A -85,B 0,C 180,E1 27201.687,E2 27201.687} C_VEL
LIN {X 0,Y 568.21,Z 51.021,A -85,B 0,C 180,E1 27198.359,E2 27198.359} C_VEL
LIN {X 0,Y 568.219,Z 51.014,A -85,B 0,C 180,E1 27195.095,E2 27195.095} C_VEL
LIN {X 0,Y 568.189,Z 51.017,A -85,B 0,C 180,E1 27191.881,E2 27191.881} C_VEL
LIN {X 0,Y 568.206,Z 51.021,A -85,B 0,C 180,E1 27188.542,E2 27188.542} C_VEL
LIN {X 0,Y 568.22,Z 51.015,A -85,B 0,C 180,E1 27185.25,E2 27185.25} C_VEL
LIN {X 0,Y 568.185,Z 51.017,A -85,B 0,C 180,E1 27182.017,E2 27182.017} C_VEL
LIN {X 0,Y 568.2,Z 51.02,A -85,B 0,C 180,E1 27178.689,E2 27178.689} C_VEL
LIN {X 0,Y 568.22,Z 51.016,A -85,B 0,C 180,E1 27175.357,E2 27175.357} C_VEL
LIN {X 0,Y 568.185,Z 51.017,A -85,B 0,C 180,E1 27172.11,E2 27172.11} C_VEL
LIN {X 0,Y 568.185,Z 51.02,A -85,B 0,C 180,E1 27168.736,E2 27168.736} C_VEL
LIN {X 0,Y 568.222,Z 51.016,A -85,B 0,C 180,E1 27165.53,E2 27165.53} C_VEL
LIN {X 0,Y 568.181,Z 51.016,A -85,B 0,C 180,E1 27162.275,E2 27162.275} C_VEL
LIN {X 0,Y 568.218,Z 51.016,A -85,B 0,C 180,E1 27159.806,E2 27159.806} C_VEL
LIN {X 0,Y 567.238,Z 51.143,A -85,B 0,C 180,E1 27159.029,E2 27159.029} C_VEL
LIN {X 0,Y 560.761,Z 51.937,A -85,B 0,C 180,E1 27156.849,E2 27156.849} C_VEL
LIN {X 0,Y 560.247,Z 51.998,A -85,B 0,C 180,E1 27156.281,E2 27156.281} C_VEL
LIN {X 0,Y 560.236,Z 52.009,A -85,B 0,C 180,E1 27152.928,E2 27152.928} C_VEL
LIN {X 0,Y 560.28,Z 52.004,A -85,B 0,C 180,E1 27149.666,E2 27149.666} C_VEL
LIN {X 0,Y 560.248,Z 52.007,A -85,B 0,C 180,E1 27146.409,E2 27146.409} C_VEL
LIN {X 0,Y 560.23,Z 52.009,A -85,B 0,C 180,E1 27143.085,E2 27143.085} C_VEL
LIN {X 0,Y 560.279,Z 52.007,A -85,B 0,C 180,E1 27139.891,E2 27139.891} C_VEL
LIN {X 0,Y 560.234,Z 52.007,A -85,B 0,C 180,E1 27136.73,E2 27136.73} C_VEL
LIN {X 0,Y 560.229,Z 52.008,A -85,B 0,C 180,E1 27133.401,E2 27133.401} C_VEL
LIN {X 0,Y 560.286,Z 52.008,A -85,B 0,C 180,E1 27130.2,E2 27130.2} C_VEL
LIN {X 0,Y 560.226,Z 52.011,A -85,B 0,C 180,E1 27126.973,E2 27126.973} C_VEL
LIN {X 0,Y 560.224,Z 52.017,A -85,B 0,C 180,E1 27123.59,E2 27123.59} C_VEL
LIN {X 0,Y 560.254,Z 52.267,A -85,B 0,C 180,E1 27123.312,E2 27123.312} C_VEL
LIN {X 0,Y 561.241,Z 58.113,A -85,B 0,C 180,E1 27122.668,E2 27122.668} C_VEL
LIN {X 0,Y 561.384,Z 87.618,A -85,B 0,C 180,E1 27119.638,E2 27119.638} C_VEL
LIN {X 0,Y 561.297,Z 117.987,A -85,B 0,C 180,E1 27116.443,E2 27116.443} C_VEL
LIN {X 0,Y 561.044,Z 148.362,A -85,B 0,C 180,E1 27113.193,E2 27113.193} C_VEL
LIN {X 0,Y 560.707,Z 176.832,A -85,B 0,C 180,E1 27110.135,E2 27110.135} C_VEL
LIN {X 0,Y 561.244,Z 183.685,A -85,B 0,C 180,E1 27110.024,E2 27110.024} C_VEL
LIN {X 0,Y 560.947,Z 287.944,A -85,B 0,C 180,E1 27108.655,E2 27108.655} C_VEL
LIN {X 0,Y 560.861,Z 302.528,A -85,B 0,C 180,E1 27108.271,E2 27108.271} C_VEL
LIN {X 0,Y 560.727,Z 315.668,A -85,B 0,C 180,E1 27107.752,E2 27107.752} C_VEL
LIN {X 0,Y 560.515,Z 330.146,A -85,B 0,C 180,E1 27106.956,E2 27106.956} C_VEL
LIN {X 0,Y 560.346,Z 343.196,A -85,B 0,C 180,E1 27106.002,E2 27106.002} C_VEL
LIN {X 0,Y 560.198,Z 354.903,A -85,B 0,C 180,E1 27104.892,E2 27104.892} C_VEL
LIN {X 0,Y 560.082,Z 364.488,A -85,B 0,C 180,E1 27103.734,E2 27103.734} C_VEL
LIN {X 0,Y 560.001,Z 372.692,A -85,B 0,C 180,E1 27102.476,E2 27102.476} C_VEL
LIN {X 0,Y 559.948,Z 379.875,A -85,B 0,C 180,E1 27101.014,E2 27101.014} C_VEL
LIN {X 0,Y 559.924,Z 384.94,A -85,B 0,C 180,E1 27099.558,E2 27099.558} C_VEL
LIN {X 0,Y 559.919,Z 388.203,A -85,B 0,C 180,E1 27098.109,E2 27098.109} C_VEL
LIN {X 0,Y 559.918,Z 389.856,A -85,B 0,C 180,E1 27096.562,E2 27096.562} C_VEL
LIN {X 0,Y 559.916,Z 389.643,A -85,B 0,C 180,E1 27095.019,E2 27095.019} C_VEL
LIN {X 0,Y 559.916,Z 387.828,A -85,B 0,C 180,E1 27093.583,E2 27093.583} C_VEL
LIN {X 0,Y 559.929,Z 384.051,A -85,B 0,C 180,E1 27092.046,E2 27092.046} C_VEL
LIN {X 0,Y 559.956,Z 378.582,A -85,B 0,C 180,E1 27090.6,E2 27090.6} C_VEL
LIN {X 0,Y 560.008,Z 371.797,A -85,B 0,C 180,E1 27089.283,E2 27089.283} C_VEL
LIN {X 0,Y 560.102,Z 362.837,A -85,B 0,C 180,E1 27087.953,E2 27087.953} C_VEL
LIN {X 0,Y 560.237,Z 352.109,A -85,B 0,C 180,E1 27086.725,E2 27086.725} C_VEL
LIN {X 0,Y 560.373,Z 339.993,A -85,B 0,C 180,E1 27085.65,E2 27085.65} C_VEL
LIN {X 0,Y 560.553,Z 327.283,A -85,B 0,C 180,E1 27084.78,E2 27084.78} C_VEL
LIN {X 0,Y 560.733,Z 314.715,A -85,B 0,C 180,E1 27084.114,E2 27084.114} C_VEL
LIN {X 0,Y 560.837,Z 299.656,A -85,B 0,C 180,E1 27083.544,E2 27083.544} C_VEL
LIN {X 0,Y 560.931,Z 283.733,A -85,B 0,C 180,E1 27083.178,E2 27083.178} C_VEL
LIN {X 0,Y 561.032,Z 173.982,A -85,B 0,C 180,E1 27081.751,E2 27081.751} C_VEL
LIN {X 0,Y 560.958,Z 170.795,A -85,B 0,C 180,E1 27081.59,E2 27081.59} C_VEL
LIN {X 0,Y 561.34,Z 128.917,A -85,B 0,C 180,E1 27078.908,E2 27078.908} C_VEL
LIN {X 0,Y 561.77,Z 81.393,A -85,B 0,C 180,E1 27075.886,E2 27075.886} C_VEL
LIN {X 0,Y 561.641,Z 57.677,A -85,B 0,C 180,E1 27074.391,E2 27074.391} C_VEL
LIN {X 0,Y 560.302,Z 52.317,A -85,B 0,C 180,E1 27073.969,E2 27073.969} C_VEL
LIN {X 0,Y 560.278,Z 52.009,A -85,B 0,C 180,E1 27073.195,E2 27073.195} C_VEL
LIN {X 0,Y 560.31,Z 52.263,A -85,B 0,C 180,E1 27072.286,E2 27072.286} C_VEL
LIN {X 0,Y 561.715,Z 57.029,A -85,B 0,C 180,E1 27071.85,E2 27071.85} C_VEL
LIN {X 0,Y 562.537,Z 60.031,A -85,B 0,C 180,E1 27071.609,E2 27071.609} C_VEL
LIN {X 0,Y 561.767,Z 110.313,A -85,B 0,C 180,E1 27068.271,E2 27068.271} C_VEL
LIN {X 0,Y 561.077,Z 161.689,A -85,B 0,C 180,E1 27064.904,E2 27064.904} C_VEL
LIN {X 0,Y 561.03,Z 172.412,A -85,B 0,C 180,E1 27064.224,E2 27064.224} C_VEL
LIN {X 0,Y 561.319,Z 182.814,A -85,B 0,C 180,E1 27064.064,E2 27064.064} C_VEL
LIN {X 0,Y 560.982,Z 287.506,A -85,B 0,C 180,E1 27062.674,E2 27062.674} C_VEL
LIN {X 0,Y 560.893,Z 301.904,A -85,B 0,C 180,E1 27062.301,E2 27062.301} C_VEL
LIN {X 0,Y 560.72,Z 316.465,A -85,B 0,C 180,E1 27061.716,E2 27061.716} C_VEL
LIN {X 0,Y 560.518,Z 329.828,A -85,B 0,C 180,E1 27060.974,E2 27060.974} C_VEL
LIN {X 0,Y 560.368,Z 342.119,A -85,B 0,C 180,E1 27060.091,E2 27060.091} C_VEL
LIN {X 0,Y 560.206,Z 354.397,A -85,B 0,C 180,E1 27058.948,E2 27058.948} C_VEL
LIN {X 0,Y 560.083,Z 364.452,A -85,B 0,C 180,E1 27057.739,E2 27057.739} C_VEL
LIN {X 0,Y 560.001,Z 372.577,A -85,B 0,C 180,E1 27056.493,E2 27056.493} C_VEL
LIN {X 0,Y 559.949,Z 379.744,A -85,B 0,C 180,E1 27055.046,E2 27055.046} C_VEL
LIN {X 0,Y 559.925,Z 385.198,A -85,B 0,C 180,E1 27053.473,E2 27053.473} C_VEL
LIN {X 0,Y 559.918,Z 388.447,A -85,B 0,C 180,E1 27051.954,E2 27051.954} C_VEL
LIN {X 0,Y 559.917,Z 389.89,A -85,B 0,C 180,E1 27050.483,E2 27050.483} C_VEL
LIN {X 0,Y 559.914,Z 389.564,A -85,B 0,C 180,E1 27048.902,E2 27048.902} C_VEL
LIN {X 0,Y 559.919,Z 387.404,A -85,B 0,C 180,E1 27047.368,E2 27047.368} C_VEL
LIN {X 0,Y 559.93,Z 383.446,A -85,B 0,C 180,E1 27045.86,E2 27045.86} C_VEL
LIN {X 0,Y 559.964,Z 377.533,A -85,B 0,C 180,E1 27044.367,E2 27044.367} C_VEL
LIN {X 0,Y 560.028,Z 369.735,A -85,B 0,C 180,E1 27042.945,E2 27042.945} C_VEL
LIN {X 0,Y 560.12,Z 361.15,A -85,B 0,C 180,E1 27041.741,E2 27041.741} C_VEL
LIN {X 0,Y 560.257,Z 350.577,A -85,B 0,C 180,E1 27040.573,E2 27040.573} C_VEL
LIN {X 0,Y 560.416,Z 338.171,A -85,B 0,C 180,E1 27039.511,E2 27039.511} C_VEL
LIN {X 0,Y 560.611,Z 324.733,A -85,B 0,C 180,E1 27038.626,E2 27038.626} C_VEL
LIN {X 0,Y 560.791,Z 311.371,A -85,B 0,C 180,E1 27037.961,E2 27037.961} C_VEL
LIN {X 0,Y 560.948,Z 296.521,A -85,B 0,C 180,E1 27037.442,E2 27037.442} C_VEL
LIN {X 0,Y 561.046,Z 280.666,A -85,B 0,C 180,E1 27037.117,E2 27037.117} C_VEL
LIN {X 0,Y 561.158,Z 179.006,A -85,B 0,C 180,E1 27035.771,E2 27035.771} C_VEL
LIN {X 0,Y 560.676,Z 175.439,A -85,B 0,C 180,E1 27035.672,E2 27035.672} C_VEL
LIN {X 0,Y 561.079,Z 144.954,A -85,B 0,C 180,E1 27032.318,E2 27032.318} C_VEL
LIN {X 0,Y 561.657,Z 115.928,A -85,B 0,C 180,E1 27029.064,E2 27029.064} C_VEL
LIN {X 0,Y 562.228,Z 86.424,A -85,B 0,C 180,E1 27025.717,E2 27025.717} C_VEL
LIN {X 0,Y 562.762,Z 61.598,A -85,B 0,C 180,E1 27022.843,E2 27022.843} C_VEL
LIN {X 0,Y 560.276,Z 52.113,A -85,B 0,C 180,E1 27021.521,E2 27021.521} C_VEL
LIN {X 0,Y 560.278,Z 52.009,A -85,B 0,C 180,E1 27018.198,E2 27018.198} C_VEL
LIN {X 0,Y 560.232,Z 52.009,A -85,B 0,C 180,E1 27014.998,E2 27014.998} C_VEL
LIN {X 0,Y 560.261,Z 52.01,A -85,B 0,C 180,E1 27011.739,E2 27011.739} C_VEL
LIN {X 0,Y 560.262,Z 52.005,A -85,B 0,C 180,E1 27008.518,E2 27008.518} C_VEL
LIN {X 0,Y 560.226,Z 52.01,A -85,B 0,C 180,E1 27005.325,E2 27005.325} C_VEL
LIN {X 0,Y 560.268,Z 52.011,A -85,B 0,C 180,E1 27002.046,E2 27002.046} C_VEL
LIN {X 0,Y 560.244,Z 52.008,A -85,B 0,C 180,E1 26998.875,E2 26998.875} C_VEL
LIN {X 0,Y 560.223,Z 52.01,A -85,B 0,C 180,E1 26995.599,E2 26995.599} C_VEL
LIN {X 0,Y 560.282,Z 52.01,A -85,B 0,C 180,E1 26992.412,E2 26992.412} C_VEL
LIN {X 0,Y 560.229,Z 52.009,A -85,B 0,C 180,E1 26989.199,E2 26989.199} C_VEL
LIN {X 0,Y 560.22,Z 52.01,A -85,B 0,C 180,E1 26985.847,E2 26985.847} C_VEL
LIN {X 0,Y 560.278,Z 52.01,A -85,B 0,C 180,E1 26982.661,E2 26982.661} C_VEL
LIN {X 0,Y 560.217,Z 52.009,A -85,B 0,C 180,E1 26979.524,E2 26979.524} C_VEL
LIN {X 0,Y 560.216,Z 52.011,A -85,B 0,C 180,E1 26976.1,E2 26976.1} C_VEL
LIN {X 0,Y 560.277,Z 52.01,A -85,B 0,C 180,E1 26972.931,E2 26972.931} C_VEL
LIN {X 0,Y 560.212,Z 52.011,A -85,B 0,C 180,E1 26969.75,E2 26969.75} C_VEL
LIN {X 0,Y 560.216,Z 52.012,A -85,B 0,C 180,E1 26966.408,E2 26966.408} C_VEL
LIN {X 0,Y 560.26,Z 52.011,A -85,B 0,C 180,E1 26963.254,E2 26963.254} C_VEL
LIN {X 0,Y 560.201,Z 52.012,A -85,B 0,C 180,E1 26960.128,E2 26960.128} C_VEL
LIN {X 0,Y 560.253,Z 52.011,A -85,B 0,C 180,E1 26957.02,E2 26957.02} C_VEL
LIN {X 0,Y 560.218,Z 52.013,A -85,B 0,C 180,E1 26953.859,E2 26953.859} C_VEL
LIN {X 0,Y 560.212,Z 52.013,A -85,B 0,C 180,E1 26950.651,E2 26950.651} C_VEL
LIN {X 0,Y 560.271,Z 52.01,A -85,B 0,C 180,E1 26947.485,E2 26947.485} C_VEL
LIN {X 0,Y 560.212,Z 52.014,A -85,B 0,C 180,E1 26944.274,E2 26944.274} C_VEL
LIN {X 0,Y 560.27,Z 52.248,A -85,B 0,C 180,E1 26941.96,E2 26941.96} C_VEL
LIN {X 0,Y 563.857,Z 63.131,A -85,B 0,C 180,E1 26940.879,E2 26940.879} C_VEL
LIN {X 0,Y 563.26,Z 97.855,A -85,B 0,C 180,E1 26938.344,E2 26938.344} C_VEL
LIN {X 0,Y 562.704,Z 144.242,A -85,B 0,C 180,E1 26935.091,E2 26935.091} C_VEL
LIN {X 0,Y 562.58,Z 158.31,A -85,B 0,C 180,E1 26934.137,E2 26934.137} C_VEL
LIN {X 0,Y 563.437,Z 166.125,A -85,B 0,C 180,E1 26934.002,E2 26934.002} C_VEL
LIN {X 0,Y 562.909,Z 366.11,A -85,B 0,C 180,E1 26931.377,E2 26931.377} C_VEL
LIN {X 0,Y 562.685,Z 385.356,A -85,B 0,C 180,E1 26930.933,E2 26930.933} C_VEL
LIN {X 0,Y 562.402,Z 403.081,A -85,B 0,C 180,E1 26930.339,E2 26930.339} C_VEL
LIN {X 0,Y 562.055,Z 421.016,A -85,B 0,C 180,E1 26929.539,E2 26929.539} C_VEL
LIN {X 0,Y 561.689,Z 437.944,A -85,B 0,C 180,E1 26928.581,E2 26928.581} C_VEL
LIN {X 0,Y 561.33,Z 453.738,A -85,B 0,C 180,E1 26927.483,E2 26927.483} C_VEL
LIN {X 0,Y 560.974,Z 468.993,A -85,B 0,C 180,E1 26926.197,E2 26926.197} C_VEL
LIN {X 0,Y 560.663,Z 483.014,A -85,B 0,C 180,E1 26924.775,E2 26924.775} C_VEL
LIN {X 0,Y 560.405,Z 495.91,A -85,B 0,C 180,E1 26923.202,E2 26923.202} C_VEL
LIN {X 0,Y 560.197,Z 507.329,A -85,B 0,C 180,E1 26921.515,E2 26921.515} C_VEL
LIN {X 0,Y 560.066,Z 516.99,A -85,B 0,C 180,E1 26919.765,E2 26919.765} C_VEL
LIN {X 0,Y 559.983,Z 524.771,A -85,B 0,C 180,E1 26918.006,E2 26918.006} C_VEL
LIN {X 0,Y 559.937,Z 531.11,A -85,B 0,C 180,E1 26916.151,E2 26916.151} C_VEL
LIN {X 0,Y 559.913,Z 535.876,A -85,B 0,C 180,E1 26914.199,E2 26914.199} C_VEL
LIN {X 0,Y 559.913,Z 538.792,A -85,B 0,C 180,E1 26912.252,E2 26912.252} C_VEL
LIN {X 0,Y 559.908,Z 539.939,A -85,B 0,C 180,E1 26910.308,E2 26910.308} C_VEL
LIN {X 0,Y 559.913,Z 539.416,A -85,B 0,C 180,E1 26908.466,E2 26908.466} C_VEL
LIN {X 0,Y 559.909,Z 537.164,A -85,B 0,C 180,E1 26906.52,E2 26906.52} C_VEL
LIN {X 0,Y 559.928,Z 533.352,A -85,B 0,C 180,E1 26904.673,E2 26904.673} C_VEL
LIN {X 0,Y 559.955,Z 527.822,A -85,B 0,C 180,E1 26902.821,E2 26902.821} C_VEL
LIN {X 0,Y 560.03,Z 520.431,A -85,B 0,C 180,E1 26900.962,E2 26900.962} C_VEL
LIN {X 0,Y 560.137,Z 511.522,A -85,B 0,C 180,E1 26899.198,E2 26899.198} C_VEL
LIN {X 0,Y 560.307,Z 501.159,A -85,B 0,C 180,E1 26897.531,E2 26897.531} C_VEL
LIN {X 0,Y 560.533,Z 489.36,A -85,B 0,C 180,E1 26895.961,E2 26895.961} C_VEL
LIN {X 0,Y 560.823,Z 475.797,A -85,B 0,C 180,E1 26894.459,E2 26894.459} C_VEL
LIN {X 0,Y 561.159,Z 461.03,A -85,B 0,C 180,E1 26893.1,E2 26893.1} C_VEL
LIN {X 0,Y 561.528,Z 445.25,A -85,B 0,C 180,E1 26891.899,E2 26891.899} C_VEL
LIN {X 0,Y 561.902,Z 428.081,A -85,B 0,C 180,E1 26890.835,E2 26890.835} C_VEL
LIN {X 0,Y 562.254,Z 410.845,A -85,B 0,C 180,E1 26889.983,E2 26889.983} C_VEL
LIN {X 0,Y 562.571,Z 392.565,A -85,B 0,C 180,E1 26889.288,E2 26889.288} C_VEL
LIN {X 0,Y 562.821,Z 373.996,A -85,B 0,C 180,E1 26888.783,E2 26888.783} C_VEL
LIN {X 0,Y 562.972,Z 353.924,A -85,B 0,C 180,E1 26888.441,E2 26888.441} C_VEL
LIN {X 0,Y 563.324,Z 157.957,A -85,B 0,C 180,E1 26885.878,E2 26885.878} C_VEL
LIN {X 0,Y 563.113,Z 153.36,A -85,B 0,C 180,E1 26885.758,E2 26885.758} C_VEL
LIN {X 0,Y 563.79,Z 76.129,A -85,B 0,C 180,E1 26882.572,E2 26882.572} C_VEL
LIN {X 0,Y 563.908,Z 62.155,A -85,B 0,C 180,E1 26881.976,E2 26881.976} C_VEL
LIN {X 0,Y 560.357,Z 52.518,A -85,B 0,C 180,E1 26881.346,E2 26881.346} C_VEL
LIN {X 0,Y 560.271,Z 52.02,A -85,B 0,C 180,E1 26881.192,E2 26881.192} C_VEL
LIN {X 0,Y 560.272,Z 52.01,A -85,B 0,C 180,E1 26877.874,E2 26877.874} C_VEL
LIN {X 0,Y 560.275,Z 52.003,A -85,B 0,C 180,E1 26874.466,E2 26874.466} C_VEL
LIN {X 0,Y 560.263,Z 52.007,A -85,B 0,C 180,E1 26871.217,E2 26871.217} C_VEL
LIN {X 0,Y 560.278,Z 52.01,A -85,B 0,C 180,E1 26867.858,E2 26867.858} C_VEL
LIN {X 0,Y 560.274,Z 52.005,A -85,B 0,C 180,E1 26864.454,E2 26864.454} C_VEL
LIN {X 0,Y 560.264,Z 52.003,A -85,B 0,C 180,E1 26861.142,E2 26861.142} C_VEL
LIN {X 0,Y 560.265,Z 52.009,A -85,B 0,C 180,E1 26857.743,E2 26857.743} C_VEL
LIN {X 0,Y 560.275,Z 52.005,A -85,B 0,C 180,E1 26854.452,E2 26854.452} C_VEL
LIN {X 0,Y 560.275,Z 52.001,A -85,B 0,C 180,E1 26851.066,E2 26851.066} C_VEL
LIN {X 0,Y 560.255,Z 52.005,A -85,B 0,C 180,E1 26847.729,E2 26847.729} C_VEL
LIN {X 0,Y 560.279,Z 52.01,A -85,B 0,C 180,E1 26844.458,E2 26844.458} C_VEL
LIN {X 0,Y 560.283,Z 52.003,A -85,B 0,C 180,E1 26841.02,E2 26841.02} C_VEL
LIN {X 0,Y 560.25,Z 52.006,A -85,B 0,C 180,E1 26837.769,E2 26837.769} C_VEL
LIN {X 0,Y 560.273,Z 52.008,A -85,B 0,C 180,E1 26834.468,E2 26834.468} C_VEL
LIN {X 0,Y 560.28,Z 52.005,A -85,B 0,C 180,E1 26831.112,E2 26831.112} C_VEL
LIN {X 0,Y 560.252,Z 52.005,A -85,B 0,C 180,E1 26827.795,E2 26827.795} C_VEL
LIN {X 0,Y 560.252,Z 52.007,A -85,B 0,C 180,E1 26824.401,E2 26824.401} C_VEL
LIN {X 0,Y 560.282,Z 52.007,A -85,B 0,C 180,E1 26821.125,E2 26821.125} C_VEL
LIN {X 0,Y 560.256,Z 52.004,A -85,B 0,C 180,E1 26817.852,E2 26817.852} C_VEL
LIN {X 0,Y 560.243,Z 52.007,A -85,B 0,C 180,E1 26814.469,E2 26814.469} C_VEL
LIN {X 0,Y 560.281,Z 52.008,A -85,B 0,C 180,E1 26811.275,E2 26811.275} C_VEL
LIN {X 0,Y 560.259,Z 52.005,A -85,B 0,C 180,E1 26807.946,E2 26807.946} C_VEL
LIN {X 0,Y 560.241,Z 52.008,A -85,B 0,C 180,E1 26804.684,E2 26804.684} C_VEL
LIN {X 0,Y 560.28,Z 52.009,A -85,B 0,C 180,E1 26801.366,E2 26801.366} C_VEL
LIN {X 0,Y 560.258,Z 52.004,A -85,B 0,C 180,E1 26798.1,E2 26798.1} C_VEL
LIN {X 0,Y 560.247,Z 51.998,A -85,B 0,C 180,E1 26796.281,E2 26796.281} C_VEL
LIN {X 0,Y 559.284,Z 52.128,A -85,B 0,C 180,E1 26795.493,E2 26795.493} C_VEL
LIN {X 0,Y 552.827,Z 52.936,A -85,B 0,C 180,E1 26793.281,E2 26793.281} C_VEL
LIN {X 0,Y 552.294,Z 52.997,A -85,B 0,C 180,E1 26792.704,E2 26792.704} C_VEL
LIN {X 0,Y 552.321,Z 52.996,A -85,B 0,C 180,E1 26789.423,E2 26789.423} C_VEL
LIN {X 0,Y 552.336,Z 52.995,A -85,B 0,C 180,E1 26786.113,E2 26786.113} C_VEL
LIN {X 0,Y 552.289,Z 52.998,A -85,B 0,C 180,E1 26782.925,E2 26782.925} C_VEL
LIN {X 0,Y 552.319,Z 52.998,A -85,B 0,C 180,E1 26779.65,E2 26779.65} C_VEL
LIN {X 0,Y 552.326,Z 52.995,A -85,B 0,C 180,E1 26776.392,E2 26776.392} C_VEL
LIN {X 0,Y 552.285,Z 52.996,A -85,B 0,C 180,E1 26773.147,E2 26773.147} C_VEL
LIN {X 0,Y 552.317,Z 53.002,A -85,B 0,C 180,E1 26769.853,E2 26769.853} C_VEL
LIN {X 0,Y 552.309,Z 52.999,A -85,B 0,C 180,E1 26766.68,E2 26766.68} C_VEL
LIN {X 0,Y 552.31,Z 53.204,A -85,B 0,C 180,E1 26763.541,E2 26763.541} C_VEL
LIN {X 0,Y 553.529,Z 59.728,A -85,B 0,C 180,E1 26762.812,E2 26762.812} C_VEL
LIN {X 0,Y 553.656,Z 90.305,A -85,B 0,C 180,E1 26759.657,E2 26759.657} C_VEL
LIN {X 0,Y 553.53,Z 120.742,A -85,B 0,C 180,E1 26756.439,E2 26756.439} C_VEL
LIN {X 0,Y 553.265,Z 151.528,A -85,B 0,C 180,E1 26753.144,E2 26753.144} C_VEL
LIN {X 0,Y 552.991,Z 177.837,A -85,B 0,C 180,E1 26750.336,E2 26750.336} C_VEL
LIN {X 0,Y 553.513,Z 184.53,A -85,B 0,C 180,E1 26750.227,E2 26750.227} C_VEL
LIN {X 0,Y 553.179,Z 288.874,A -85,B 0,C 180,E1 26748.838,E2 26748.838} C_VEL
